KUKA KRL program: EPS_2_25694_LG05A_A_20260223033046.src

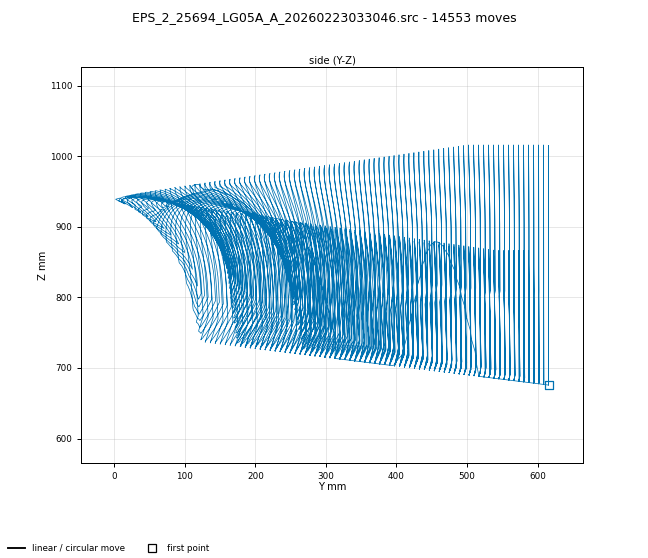
[picture p0: tool path of EPS_2_25694_LG05A_A_20260223033046.src, 14553 of 14555 moves have a stored position in this frame; points joined in program order, loops and branches not executed]
&ACCESS RVP
&REL 4
&COMMENT QRS 19112012
&PARAM EDITMASK = *
DEF PART()
EXT BAS (BAS_COMMAND :IN,REAL :IN )
INT I
BAS (#INITMOV,0 )

;KUKA QRS Post kuka4.cps  Date:22-06-2017 !

File_ID=3044

QRS_PRE_INIT()

;Init var - Until changes are made in qrs_pre_init
Outlet_Square_prg=0
Inlet_1_Square_prg=0
Inlet_2_Square_prg=0
Inlet_3_Square_prg=0
Inlet_4_Square_prg=0
Inlet_5_Square_prg=0

Outlet_1={X 0.000, Y 502.870, Z 915.500, B 0.000, E1 0.000 }
Inlet_1={X 0.000, Y 543.190, Z 350.500, B 0.000, E1 155.000 }
Inlet_2={X 0.000, Y 517.510, Z 710.500, B 0.000, E1 257.000 }
Outlet_1_type=201
Inlet_1_type=201
Inlet_2_type=201
;QRS#1=Sidecore dimensions
;QRS#2=200-8" PVC SDR 35
;QRS#3=200-8" PVC SDR 35
;QRS#4=200-8" PVC SDR 35
;QRS#5=
;QRS#6=
;QRS#7=
;QRS#8=
;QRS#9=12-08 PSX
;QRS#10=12-08 PSX
;QRS#11=12-08 PSX
;QRS#12=
;QRS#13=
;QRS#14=
;QRS#15=
;QRS#16=1220x127x1295 4,25'
;QRS#17=EPS Height
;QRS#18=1016
;QRS#19=*
;QRS#20= UPDATED VERSION 22-06-2017
;QRS#21=*
Outlet_Square=0100
Inlet_1_Square=0100
Inlet_2_Square=0100
Inlet_3_Square=0
Inlet_4_Square=0
Inlet_5_Square=0
Mill_Square=1
Outlet_Square_Prg=204
Inlet_1_Square_prg=204
Inlet_2_Square_prg=204

QRS_INIT()

$ADVANCE=5

; T1
PTP {E1 173.41,E2 173.41}
PTP {X 0,Y 615.487,A -85,B 0,C 180,E1 173.41,E2 173.41,E3 0,E4 0,E5 0,E6 0}
QRS_SPEED_INIT()
LIN {X 0,Y 615.487,Z 675.703,A -85,B 0,C 180,E1 173.41,E2 173.41,E3 0,E4 0,E5 0,E6 0} C_VEL
LIN {X 0,Y 615.494,Z 675.684,A -85,B 0,C 180,E1 170.801,E2 170.801} C_VEL
LIN {X 0,Y 615.457,Z 675.687,A -85,B 0,C 180,E1 168.138,E2 168.138} C_VEL
LIN {X 0,Y 615.465,Z 675.696,A -85,B 0,C 180,E1 165.45,E2 165.45} C_VEL
LIN {X 0,Y 615.489,Z 675.691,A -85,B 0,C 180,E1 162.729,E2 162.729} C_VEL
LIN {X 0,Y 615.462,Z 675.686,A -85,B 0,C 180,E1 159.966,E2 159.966} C_VEL
LIN {X 0,Y 615.452,Z 675.689,A -85,B 0,C 180,E1 157.659,E2 157.659} C_VEL
LIN {X 0,Y 615.47,Z 675.697,A -85,B 0,C 180,E1 155.007,E2 155.007} C_VEL
LIN {X 0,Y 615.484,Z 675.685,A -85,B 0,C 180,E1 152.084,E2 152.084} C_VEL
LIN {X 0,Y 615.481,Z 675.683,A -85,B 0,C 180,E1 149.839,E2 149.839} C_VEL
LIN {X 0,Y 615.46,Z 675.686,A -85,B 0,C 180,E1 147.541,E2 147.541} C_VEL
LIN {X 0,Y 615.448,Z 675.69,A -85,B 0,C 180,E1 145.182,E2 145.182} C_VEL
LIN {X 0,Y 615.456,Z 675.694,A -85,B 0,C 180,E1 142.755,E2 142.755} C_VEL
LIN {X 0,Y 615.49,Z 675.691,A -85,B 0,C 180,E1 139.909,E2 139.909} C_VEL
LIN {X 0,Y 615.497,Z 675.684,A -85,B 0,C 180,E1 137.647,E2 137.647} C_VEL
LIN {X 0,Y 615.449,Z 675.689,A -85,B 0,C 180,E1 134.927,E2 134.927} C_VEL
LIN {X 0,Y 615.476,Z 675.699,A -85,B 0,C 180,E1 132.078,E2 132.078} C_VEL
LIN {X 0,Y 615.466,Z 675.686,A -85,B 0,C 180,E1 129.059,E2 129.059} C_VEL
LIN {X 0,Y 615.496,Z 675.783,A -85,B 0,C 180,E1 127.719,E2 127.719} C_VEL
LIN {X 0,Y 615.495,Z 676.753,A -85,B 0,C 180,E1 127.575,E2 127.575} C_VEL
LIN {X 0,Y 615.499,Z 708.482,A -85,B 0,C 180,E1 127.183,E2 127.183} C_VEL
LIN {X 0,Y 615.497,Z 761.445,A -85,B 0,C 180,E1 126.551,E2 126.551} C_VEL
LIN {X 0,Y 615.5,Z 774.268,A -85,B 0,C 180,E1 126.275,E2 126.275} C_VEL
LIN {X 0,Y 615.5,Z 785.845,A -85,B 0,C 180,E1 125.908,E2 125.908} C_VEL
LIN {X 0,Y 615.495,Z 798.517,A -85,B 0,C 180,E1 125.363,E2 125.363} C_VEL
LIN {X 0,Y 615.485,Z 810.253,A -85,B 0,C 180,E1 124.7,E2 124.7} C_VEL
LIN {X 0,Y 615.497,Z 821.428,A -85,B 0,C 180,E1 123.898,E2 123.898} C_VEL
LIN {X 0,Y 615.497,Z 828.942,A -85,B 0,C 180,E1 123.234,E2 123.234} C_VEL
LIN {X 0,Y 615.496,Z 837.643,A -85,B 0,C 180,E1 122.331,E2 122.331} C_VEL
LIN {X 0,Y 615.493,Z 844.95,A -85,B 0,C 180,E1 121.385,E2 121.385} C_VEL
LIN {X 0,Y 615.495,Z 851.375,A -85,B 0,C 180,E1 120.348,E2 120.348} C_VEL
LIN {X 0,Y 615.498,Z 856.021,A -85,B 0,C 180,E1 119.404,E2 119.404} C_VEL
LIN {X 0,Y 615.496,Z 859.685,A -85,B 0,C 180,E1 118.451,E2 118.451} C_VEL
LIN {X 0,Y 615.496,Z 863.106,A -85,B 0,C 180,E1 117.175,E2 117.175} C_VEL
LIN {X 0,Y 615.493,Z 864.37,A -85,B 0,C 180,E1 116.443,E2 116.443} C_VEL
LIN {X 0,Y 615.496,Z 865.202,A -85,B 0,C 180,E1 115.569,E2 115.569} C_VEL
LIN {X 0,Y 615.494,Z 865.386,A -85,B 0,C 180,E1 114.99,E2 114.99} C_VEL
LIN {X 0,Y 615.496,Z 864.968,A -85,B 0,C 180,E1 114.009,E2 114.009} C_VEL
LIN {X 0,Y 615.496,Z 863.341,A -85,B 0,C 180,E1 112.843,E2 112.843} C_VEL
LIN {X 0,Y 615.495,Z 860.72,A -85,B 0,C 180,E1 111.782,E2 111.782} C_VEL
LIN {X 0,Y 615.497,Z 856.247,A -85,B 0,C 180,E1 110.558,E2 110.558} C_VEL
LIN {X 0,Y 615.496,Z 850.128,A -85,B 0,C 180,E1 109.336,E2 109.336} C_VEL
LIN {X 0,Y 615.494,Z 843.188,A -85,B 0,C 180,E1 108.28,E2 108.28} C_VEL
LIN {X 0,Y 615.498,Z 834.872,A -85,B 0,C 180,E1 107.269,E2 107.269} C_VEL
LIN {X 0,Y 615.498,Z 824.879,A -85,B 0,C 180,E1 106.3,E2 106.3} C_VEL
LIN {X 0,Y 615.491,Z 814.314,A -85,B 0,C 180,E1 105.479,E2 105.479} C_VEL
LIN {X 0,Y 615.488,Z 803.371,A -85,B 0,C 180,E1 104.802,E2 104.802} C_VEL
LIN {X 0,Y 615.498,Z 791.85,A -85,B 0,C 180,E1 104.241,E2 104.241} C_VEL
LIN {X 0,Y 615.496,Z 779.587,A -85,B 0,C 180,E1 103.789,E2 103.789} C_VEL
LIN {X 0,Y 615.498,Z 766.533,A -85,B 0,C 180,E1 103.452,E2 103.452} C_VEL
LIN {X 0,Y 615.5,Z 750.675,A -85,B 0,C 180,E1 103.221,E2 103.221} C_VEL
LIN {X 0,Y 615.498,Z 676.849,A -85,B 0,C 180,E1 102.34,E2 102.34} C_VEL
LIN {X 0,Y 615.493,Z 675.917,A -85,B 0,C 180,E1 102.236,E2 102.236} C_VEL
LIN {X 0,Y 615.473,Z 675.691,A -85,B 0,C 180,E1 100.526,E2 100.526} C_VEL
LIN {X 0,Y 615.478,Z 675.7,A -85,B 0,C 180,E1 97.875,E2 97.875} C_VEL
LIN {X 0,Y 615.428,Z 675.696,A -85,B 0,C 180,E1 95.241,E2 95.241} C_VEL
LIN {X 0,Y 615.432,Z 675.697,A -85,B 0,C 180,E1 93.272,E2 93.272} C_VEL
LIN {X 0,Y 615.439,Z 675.697,A -85,B 0,C 180,E1 91.308,E2 91.308} C_VEL
LIN {X 0,Y 615.447,Z 675.698,A -85,B 0,C 180,E1 89.345,E2 89.345} C_VEL
LIN {X 0,Y 615.457,Z 675.698,A -85,B 0,C 180,E1 87.381,E2 87.381} C_VEL
LIN {X 0,Y 615.422,Z 675.696,A -85,B 0,C 180,E1 84.757,E2 84.757} C_VEL
LIN {X 0,Y 615.424,Z 675.696,A -85,B 0,C 180,E1 82.783,E2 82.783} C_VEL
LIN {X 0,Y 615.426,Z 675.697,A -85,B 0,C 180,E1 80.799,E2 80.799} C_VEL
LIN {X 0,Y 615.429,Z 675.697,A -85,B 0,C 180,E1 78.805,E2 78.805} C_VEL
LIN {X 0,Y 615.429,Z 675.698,A -85,B 0,C 180,E1 76.797,E2 76.797} C_VEL
LIN {X 0,Y 615.435,Z 675.698,A -85,B 0,C 180,E1 74.772,E2 74.772} C_VEL
LIN {X 0,Y 615.436,Z 675.698,A -85,B 0,C 180,E1 72.727,E2 72.727} C_VEL
LIN {X 0,Y 615.435,Z 675.698,A -85,B 0,C 180,E1 70.659,E2 70.659} C_VEL
LIN {X 0,Y 615.433,Z 675.698,A -85,B 0,C 180,E1 68.565,E2 68.565} C_VEL
LIN {X 0,Y 615.427,Z 675.698,A -85,B 0,C 180,E1 66.44,E2 66.44} C_VEL
LIN {X 0,Y 615.421,Z 675.698,A -85,B 0,C 180,E1 64.28,E2 64.28} C_VEL
LIN {X 0,Y 615.417,Z 675.697,A -85,B 0,C 180,E1 62.081,E2 62.081} C_VEL
LIN {X 0,Y 615.415,Z 675.697,A -85,B 0,C 180,E1 59.835,E2 59.835} C_VEL
LIN {X 0,Y 615.425,Z 675.696,A -85,B 0,C 180,E1 57.538,E2 57.538} C_VEL
LIN {X 0,Y 615.449,Z 675.695,A -85,B 0,C 180,E1 55.182,E2 55.182} C_VEL
LIN {X 0,Y 615.489,Z 675.697,A -85,B 0,C 180,E1 52.757,E2 52.757} C_VEL
LIN {X 0,Y 615.425,Z 675.698,A -85,B 0,C 180,E1 49.918,E2 49.918} C_VEL
LIN {X 0,Y 615.415,Z 675.698,A -85,B 0,C 180,E1 47.64,E2 47.64} C_VEL
LIN {X 0,Y 615.439,Z 675.696,A -85,B 0,C 180,E1 44.926,E2 44.926} C_VEL
LIN {X 0,Y 615.467,Z 675.699,A -85,B 0,C 180,E1 42.077,E2 42.077} C_VEL
LIN {X 0,Y 615.436,Z 675.699,A -85,B 0,C 180,E1 39.755,E2 39.755} C_VEL
LIN {X 0,Y 615.41,Z 675.698,A -85,B 0,C 180,E1 37.248,E2 37.248} C_VEL
LIN {X 0,Y 615.428,Z 675.697,A -85,B 0,C 180,E1 34.691,E2 34.691} C_VEL
LIN {X 0,Y 615.46,Z 675.696,A -85,B 0,C 180,E1 32.325,E2 32.325} C_VEL
LIN {X 0,Y 615.432,Z 675.699,A -85,B 0,C 180,E1 29.409,E2 29.409} C_VEL
LIN {X 0,Y 615.412,Z 675.699,A -85,B 0,C 180,E1 27.03,E2 27.03} C_VEL
LIN {X 0,Y 615.499,Z 675.896,A -85,B 0,C 180,E1 25.679,E2 25.679} C_VEL
LIN {X 0,Y 615.5,Z 676.846,A -85,B 0,C 180,E1 25.57,E2 25.57} C_VEL
LIN {X 0,Y 615.495,Z 761.983,A -85,B 0,C 180,E1 24.541,E2 24.541} C_VEL
LIN {X 0,Y 615.498,Z 775.58,A -85,B 0,C 180,E1 24.239,E2 24.239} C_VEL
LIN {X 0,Y 615.497,Z 787.695,A -85,B 0,C 180,E1 23.839,E2 23.839} C_VEL
LIN {X 0,Y 615.493,Z 799.977,A -85,B 0,C 180,E1 23.289,E2 23.289} C_VEL
LIN {X 0,Y 615.485,Z 811.851,A -85,B 0,C 180,E1 22.595,E2 22.595} C_VEL
LIN {X 0,Y 615.498,Z 821.768,A -85,B 0,C 180,E1 21.872,E2 21.872} C_VEL
LIN {X 0,Y 615.499,Z 830.51,A -85,B 0,C 180,E1 21.081,E2 21.081} C_VEL
LIN {X 0,Y 615.496,Z 837.947,A -85,B 0,C 180,E1 20.295,E2 20.295} C_VEL
LIN {X 0,Y 615.497,Z 845.264,A -85,B 0,C 180,E1 19.338,E2 19.338} C_VEL
LIN {X 0,Y 615.498,Z 851.739,A -85,B 0,C 180,E1 18.281,E2 18.281} C_VEL
LIN {X 0,Y 615.495,Z 856.597,A -85,B 0,C 180,E1 17.27,E2 17.27} C_VEL
LIN {X 0,Y 615.495,Z 859.748,A -85,B 0,C 180,E1 16.431,E2 16.431} C_VEL
LIN {X 0,Y 615.496,Z 862.997,A -85,B 0,C 180,E1 15.226,E2 15.226} C_VEL
LIN {X 0,Y 615.494,Z 864.223,A -85,B 0,C 180,E1 14.549,E2 14.549} C_VEL
LIN {X 0,Y 615.494,Z 864.987,A -85,B 0,C 180,E1 13.874,E2 13.874} C_VEL
LIN {X 0,Y 615.495,Z 865.294,A -85,B 0,C 180,E1 12.53,E2 12.53} C_VEL
LIN {X 0,Y 615.495,Z 864.834,A -85,B 0,C 180,E1 11.861,E2 11.861} C_VEL
LIN {X 0,Y 615.494,Z 863.432,A -85,B 0,C 180,E1 10.888,E2 10.888} C_VEL
LIN {X 0,Y 615.498,Z 859.912,A -85,B 0,C 180,E1 9.53,E2 9.53} C_VEL
LIN {X 0,Y 615.495,Z 856.155,A -85,B 0,C 180,E1 8.537,E2 8.537} C_VEL
LIN {X 0,Y 615.497,Z 851.282,A -85,B 0,C 180,E1 7.546,E2 7.546} C_VEL
LIN {X 0,Y 615.488,Z 845.163,A -85,B 0,C 180,E1 6.557,E2 6.557} C_VEL
LIN {X 0,Y 615.498,Z 837.565,A -85,B 0,C 180,E1 5.57,E2 5.57} C_VEL
LIN {X 0,Y 615.497,Z 828.01,A -85,B 0,C 180,E1 4.585,E2 4.585} C_VEL
LIN {X 0,Y 615.5,Z 818.276,A -85,B 0,C 180,E1 3.765,E2 3.765} C_VEL
LIN {X 0,Y 615.492,Z 807.277,A -85,B 0,C 180,E1 3.027,E2 3.027} C_VEL
LIN {X 0,Y 615.498,Z 796.564,A -85,B 0,C 180,E1 2.454,E2 2.454} C_VEL
LIN {X 0,Y 615.5,Z 784.792,A -85,B 0,C 180,E1 1.963,E2 1.963} C_VEL
LIN {X 0,Y 615.498,Z 772.808,A -85,B 0,C 180,E1 1.595,E2 1.595} C_VEL
LIN {X 0,Y 615.499,Z 760.801,A -85,B 0,C 180,E1 1.35,E2 1.35} C_VEL
LIN {X 0,Y 615.497,Z 677.006,A -85,B 0,C 180,E1 0.348,E2 0.348} C_VEL
LIN {X 0,Y 615.498,Z 675.959,A -85,B 0,C 180,E1 0.245,E2 0.245} C_VEL
LIN {X 0,Y 615.469,Z 675.686,A -85,B 0,C 180,E1 -0.654,E2 -0.654} C_VEL
LIN {X 0,Y 615.489,Z 675.682,A -85,B 0,C 180,E1 -3.273,E2 -3.273} C_VEL
LIN {X 0,Y 615.488,Z 675.696,A -85,B 0,C 180,E1 -5.898,E2 -5.898} C_VEL
LIN {X 0,Y 615.471,Z 675.693,A -85,B 0,C 180,E1 -8.537,E2 -8.537} C_VEL
LIN {X 0,Y 615.483,Z 675.681,A -85,B 0,C 180,E1 -11.193,E2 -11.193} C_VEL
LIN {X 0,Y 615.482,Z 675.69,A -85,B 0,C 180,E1 -13.928,E2 -13.928} C_VEL
LIN {X 0,Y 615.48,Z 675.697,A -85,B 0,C 180,E1 -16.587,E2 -16.587} C_VEL
LIN {X 0,Y 615.474,Z 675.684,A -85,B 0,C 180,E1 -19.338,E2 -19.338} C_VEL
LIN {X 0,Y 615.482,Z 675.689,A -85,B 0,C 180,E1 -22.137,E2 -22.137} C_VEL
LIN {X 0,Y 615.473,Z 675.694,A -85,B 0,C 180,E1 -24.992,E2 -24.992} C_VEL
LIN {X 0,Y 615.468,Z 675.692,A -85,B 0,C 180,E1 -27.178,E2 -27.178} C_VEL
LIN {X 0,Y 615.481,Z 675.682,A -85,B 0,C 180,E1 -29.792,E2 -29.792} C_VEL
LIN {X 0,Y 615.481,Z 675.688,A -85,B 0,C 180,E1 -32.458,E2 -32.458} C_VEL
LIN {X 0,Y 615.488,Z 675.696,A -85,B 0,C 180,E1 -34.815,E2 -34.815} C_VEL
LIN {X 0,Y 615.479,Z 675.698,A -85,B 0,C 180,E1 -37.243,E2 -37.243} C_VEL
LIN {X 0,Y 615.475,Z 675.683,A -85,B 0,C 180,E1 -40.087,E2 -40.087} C_VEL
LIN {X 0,Y 615.487,Z 675.695,A -85,B 0,C 180,E1 -43.046,E2 -43.046} C_VEL
LIN {X 0,Y 615.466,Z 675.688,A -85,B 0,C 180,E1 -46.005,E2 -46.005} C_VEL
LIN {X 0,Y 615.485,Z 675.686,A -85,B 0,C 180,E1 -48.906,E2 -48.906} C_VEL
LIN {X 0,Y 615.482,Z 675.689,A -85,B 0,C 180,E1 -51.094,E2 -51.094} C_VEL
LIN {X 0,Y 615.484,Z 675.703,A -85,B 0,C 180,E1 -53.574,E2 -53.574} C_VEL
LIN {X 0,Y 615.473,Z 675.695,A -85,B 0,C 180,E1 -55.976,E2 -55.976} C_VEL
LIN {X 0,Y 615.464,Z 675.69,A -85,B 0,C 180,E1 -58.312,E2 -58.312} C_VEL
LIN {X 0,Y 615.467,Z 675.686,A -85,B 0,C 180,E1 -60.592,E2 -60.592} C_VEL
LIN {X 0,Y 615.485,Z 675.681,A -85,B 0,C 180,E1 -62.956,E2 -62.956} C_VEL
LIN {X 0,Y 615.497,Z 675.933,A -85,B 0,C 180,E1 -64.057,E2 -64.057} C_VEL
LIN {X 0,Y 615.472,Z 692.484,A -85,B 0,C 180,E1 -65.863,E2 -65.863} C_VEL
LIN {X 0,Y 615.448,Z 716.422,A -85,B 0,C 180,E1 -68.39,E2 -68.39} C_VEL
LIN {X 0,Y 615.482,Z 743.317,A -85,B 0,C 180,E1 -71.18,E2 -71.18} C_VEL
LIN {X 0,Y 615.458,Z 771.867,A -85,B 0,C 180,E1 -74.093,E2 -74.093} C_VEL
LIN {X 0,Y 615.477,Z 798.699,A -85,B 0,C 180,E1 -76.798,E2 -76.798} C_VEL
LIN {X 0,Y 615.495,Z 801.848,A -85,B 0,C 180,E1 -77.092,E2 -77.092} C_VEL
LIN {X 0,Y 615.483,Z 911.78,A -85,B 0,C 180,E1 -78.41,E2 -78.41} C_VEL
LIN {X 0,Y 615.498,Z 924.309,A -85,B 0,C 180,E1 -78.681,E2 -78.681} C_VEL
LIN {X 0,Y 615.496,Z 937.503,A -85,B 0,C 180,E1 -79.109,E2 -79.109} C_VEL
LIN {X 0,Y 615.493,Z 949.458,A -85,B 0,C 180,E1 -79.639,E2 -79.639} C_VEL
LIN {X 0,Y 615.483,Z 960.982,A -85,B 0,C 180,E1 -80.303,E2 -80.303} C_VEL
LIN {X 0,Y 615.499,Z 971.329,A -85,B 0,C 180,E1 -81.049,E2 -81.049} C_VEL
LIN {X 0,Y 615.497,Z 979.682,A -85,B 0,C 180,E1 -81.793,E2 -81.793} C_VEL
LIN {X 0,Y 615.498,Z 987.598,A -85,B 0,C 180,E1 -82.619,E2 -82.619} C_VEL
LIN {X 0,Y 615.491,Z 995.198,A -85,B 0,C 180,E1 -83.607,E2 -83.607} C_VEL
LIN {X 0,Y 615.498,Z 1002.199,A -85,B 0,C 180,E1 -84.758,E2 -84.758} C_VEL
LIN {X 0,Y 615.493,Z 1006.847,A -85,B 0,C 180,E1 -85.743,E2 -85.743} C_VEL
LIN {X 0,Y 615.494,Z 1010.396,A -85,B 0,C 180,E1 -86.726,E2 -86.726} C_VEL
LIN {X 0,Y 615.497,Z 1012.23,A -85,B 0,C 180,E1 -87.381,E2 -87.381} C_VEL
LIN {X 0,Y 615.497,Z 1013.607,A -85,B 0,C 180,E1 -88.036,E2 -88.036} C_VEL
LIN {X 0,Y 615.496,Z 1015.173,A -85,B 0,C 180,E1 -89.345,E2 -89.345} C_VEL
LIN {X 0,Y 615.494,Z 1015.389,A -85,B 0,C 180,E1 -89.999,E2 -89.999} C_VEL
LIN {X 0,Y 615.495,Z 1014.581,A -85,B 0,C 180,E1 -91.308,E2 -91.308} C_VEL
LIN {X 0,Y 615.497,Z 1013.61,A -85,B 0,C 180,E1 -91.962,E2 -91.962} C_VEL
LIN {X 0,Y 615.497,Z 1012.235,A -85,B 0,C 180,E1 -92.617,E2 -92.617} C_VEL
LIN {X 0,Y 615.496,Z 1009.353,A -85,B 0,C 180,E1 -93.6,E2 -93.6} C_VEL
LIN {X 0,Y 615.498,Z 1005.446,A -85,B 0,C 180,E1 -94.583,E2 -94.583} C_VEL
LIN {X 0,Y 615.499,Z 1000.41,A -85,B 0,C 180,E1 -95.569,E2 -95.569} C_VEL
LIN {X 0,Y 615.49,Z 993.913,A -85,B 0,C 180,E1 -96.578,E2 -96.578} C_VEL
LIN {X 0,Y 615.497,Z 986.142,A -85,B 0,C 180,E1 -97.544,E2 -97.544} C_VEL
LIN {X 0,Y 615.498,Z 976.269,A -85,B 0,C 180,E1 -98.535,E2 -98.535} C_VEL
LIN {X 0,Y 615.495,Z 965.88,A -85,B 0,C 180,E1 -99.363,E2 -99.363} C_VEL
LIN {X 0,Y 615.482,Z 955.594,A -85,B 0,C 180,E1 -100.027,E2 -100.027} C_VEL
LIN {X 0,Y 615.497,Z 944.112,A -85,B 0,C 180,E1 -100.617,E2 -100.617} C_VEL
LIN {X 0,Y 615.499,Z 932.285,A -85,B 0,C 180,E1 -101.079,E2 -101.079} C_VEL
LIN {X 0,Y 615.494,Z 919.286,A -85,B 0,C 180,E1 -101.442,E2 -101.442} C_VEL
LIN {X 0,Y 615.479,Z 906.029,A -85,B 0,C 180,E1 -101.672,E2 -101.672} C_VEL
LIN {X 0,Y 615.495,Z 801.887,A -85,B 0,C 180,E1 -102.906,E2 -102.906} C_VEL
LIN {X 0,Y 615.439,Z 776.921,A -85,B 0,C 180,E1 -105.396,E2 -105.396} C_VEL
LIN {X 0,Y 615.495,Z 751.738,A -85,B 0,C 180,E1 -107.956,E2 -107.956} C_VEL
LIN {X 0,Y 615.492,Z 724.847,A -85,B 0,C 180,E1 -110.729,E2 -110.729} C_VEL
LIN {X 0,Y 615.444,Z 699.632,A -85,B 0,C 180,E1 -113.379,E2 -113.379} C_VEL
LIN {X 0,Y 615.494,Z 676.165,A -85,B 0,C 180,E1 -115.896,E2 -115.896} C_VEL
LIN {X 0,Y 615.498,Z 675.721,A -85,B 0,C 180,E1 -116.078,E2 -116.078} C_VEL
LIN {X 0,Y 615.485,Z 675.687,A -85,B 0,C 180,E1 -118.657,E2 -118.657} C_VEL
LIN {X 0,Y 615.482,Z 675.682,A -85,B 0,C 180,E1 -121.085,E2 -121.085} C_VEL
LIN {X 0,Y 615.467,Z 675.686,A -85,B 0,C 180,E1 -123.531,E2 -123.531} C_VEL
LIN {X 0,Y 615.462,Z 675.69,A -85,B 0,C 180,E1 -125.83,E2 -125.83} C_VEL
LIN {X 0,Y 615.462,Z 675.693,A -85,B 0,C 180,E1 -128.069,E2 -128.069} C_VEL
LIN {X 0,Y 615.488,Z 675.703,A -85,B 0,C 180,E1 -130.605,E2 -130.605} C_VEL
LIN {X 0,Y 615.489,Z 675.684,A -85,B 0,C 180,E1 -133.243,E2 -133.243} C_VEL
LIN {X 0,Y 615.463,Z 675.687,A -85,B 0,C 180,E1 -136.003,E2 -136.003} C_VEL
LIN {X 0,Y 615.468,Z 675.694,A -85,B 0,C 180,E1 -138.524,E2 -138.524} C_VEL
LIN {X 0,Y 615.492,Z 675.697,A -85,B 0,C 180,E1 -141.096,E2 -141.096} C_VEL
LIN {X 0,Y 615.489,Z 675.685,A -85,B 0,C 180,E1 -143.575,E2 -143.575} C_VEL
LIN {X 0,Y 615.487,Z 675.681,A -85,B 0,C 180,E1 -145.978,E2 -145.978} C_VEL
LIN {X 0,Y 615.466,Z 675.685,A -85,B 0,C 180,E1 -148.313,E2 -148.313} C_VEL
LIN {X 0,Y 615.459,Z 675.688,A -85,B 0,C 180,E1 -150.592,E2 -150.592} C_VEL
LIN {X 0,Y 615.463,Z 675.693,A -85,B 0,C 180,E1 -152.957,E2 -152.957} C_VEL
LIN {X 0,Y 615.489,Z 675.693,A -85,B 0,C 180,E1 -155.728,E2 -155.728} C_VEL
LIN {X 0,Y 615.471,Z 675.684,A -85,B 0,C 180,E1 -158.568,E2 -158.568} C_VEL
LIN {X 0,Y 615.469,Z 675.684,A -85,B 0,C 180,E1 -160.661,E2 -160.661} C_VEL
LIN {X 0,Y 615.465,Z 675.695,A -85,B 0,C 180,E1 -163.413,E2 -163.413} C_VEL
LIN {X 0,Y 615.488,Z 675.692,A -85,B 0,C 180,E1 -166.126,E2 -166.126} C_VEL
LIN {X 0,Y 615.479,Z 675.682,A -85,B 0,C 180,E1 -168.807,E2 -168.807} C_VEL
LIN {X 0,Y 615.456,Z 675.691,A -85,B 0,C 180,E1 -171.463,E2 -171.463} C_VEL
LIN {X 0,Y 615.494,Z 675.699,A -85,B 0,C 180,E1 -174.102,E2 -174.102} C_VEL
LIN {X 0,Y 615.492,Z 675.685,A -85,B 0,C 180,E1 -176.727,E2 -176.727} C_VEL
LIN {X 0,Y 615.461,Z 675.686,A -85,B 0,C 180,E1 -179.346,E2 -179.346} C_VEL
LIN {X 0,Y 615.458,Z 675.693,A -85,B 0,C 180,E1 -181.963,E2 -181.963} C_VEL
LIN {X 0,Y 615.497,Z 675.698,A -85,B 0,C 180,E1 -184.585,E2 -184.585} C_VEL
LIN {X 0,Y 615.487,Z 675.703,A -85,B 0,C 180,E1 -186.59,E2 -186.59} C_VEL
LIN {X 0,Y 614.814,Z 675.833,A -85,B 0,C 180,E1 -187.136,E2 -187.136} C_VEL
LIN {X 0,Y 611.988,Z 676.247,A -85,B 0,C 180,E1 -188.022,E2 -188.022} C_VEL
LIN {X 0,Y 609.594,Z 676.558,A -85,B 0,C 180,E1 -188.734,E2 -188.734} C_VEL
LIN {X 0,Y 608.548,Z 676.677,A -85,B 0,C 180,E1 -189.284,E2 -189.284} C_VEL
LIN {X 0,Y 608.452,Z 676.687,A -85,B 0,C 180,E1 -189.47,E2 -189.47} C_VEL
LIN {X 0,Y 608.437,Z 676.689,A -85,B 0,C 180,E1 -192,E2 -192} C_VEL
LIN {X 0,Y 608.461,Z 676.694,A -85,B 0,C 180,E1 -194.721,E2 -194.721} C_VEL
LIN {X 0,Y 608.447,Z 676.69,A -85,B 0,C 180,E1 -197.477,E2 -197.477} C_VEL
LIN {X 0,Y 608.435,Z 676.689,A -85,B 0,C 180,E1 -200.275,E2 -200.275} C_VEL
LIN {X 0,Y 608.447,Z 676.688,A -85,B 0,C 180,E1 -202.477,E2 -202.477} C_VEL
LIN {X 0,Y 608.446,Z 676.698,A -85,B 0,C 180,E1 -205.301,E2 -205.301} C_VEL
LIN {X 0,Y 608.442,Z 676.696,A -85,B 0,C 180,E1 -207.519,E2 -207.519} C_VEL
LIN {X 0,Y 608.451,Z 676.686,A -85,B 0,C 180,E1 -210.546,E2 -210.546} C_VEL
LIN {X 0,Y 608.437,Z 676.689,A -85,B 0,C 180,E1 -212.881,E2 -212.881} C_VEL
LIN {X 0,Y 608.434,Z 676.694,A -85,B 0,C 180,E1 -215.279,E2 -215.279} C_VEL
LIN {X 0,Y 608.466,Z 676.687,A -85,B 0,C 180,E1 -218.242,E2 -218.242} C_VEL
LIN {X 0,Y 608.419,Z 676.692,A -85,B 0,C 180,E1 -221.18,E2 -221.18} C_VEL
LIN {X 0,Y 608.466,Z 676.696,A -85,B 0,C 180,E1 -223.87,E2 -223.87} C_VEL
LIN {X 0,Y 608.464,Z 676.686,A -85,B 0,C 180,E1 -226.692,E2 -226.692} C_VEL
LIN {X 0,Y 608.443,Z 676.688,A -85,B 0,C 180,E1 -228.824,E2 -228.824} C_VEL
LIN {X 0,Y 608.448,Z 676.691,A -85,B 0,C 180,E1 -231.763,E2 -231.763} C_VEL
LIN {X 0,Y 608.505,Z 676.96,A -85,B 0,C 180,E1 -232.221,E2 -232.221} C_VEL
LIN {X 0,Y 608.596,Z 677.93,A -85,B 0,C 180,E1 -232.305,E2 -232.305} C_VEL
LIN {X 0,Y 608.563,Z 762.201,A -85,B 0,C 180,E1 -233.327,E2 -233.327} C_VEL
LIN {X 0,Y 608.547,Z 775.37,A -85,B 0,C 180,E1 -233.621,E2 -233.621} C_VEL
LIN {X 0,Y 608.526,Z 787.298,A -85,B 0,C 180,E1 -234.015,E2 -234.015} C_VEL
LIN {X 0,Y 608.518,Z 798.871,A -85,B 0,C 180,E1 -234.526,E2 -234.526} C_VEL
LIN {X 0,Y 608.474,Z 810.468,A -85,B 0,C 180,E1 -235.188,E2 -235.188} C_VEL
LIN {X 0,Y 608.472,Z 820.84,A -85,B 0,C 180,E1 -235.931,E2 -235.931} C_VEL
LIN {X 0,Y 608.475,Z 828.838,A -85,B 0,C 180,E1 -236.629,E2 -236.629} C_VEL
LIN {X 0,Y 608.473,Z 837.054,A -85,B 0,C 180,E1 -237.477,E2 -237.477} C_VEL
LIN {X 0,Y 608.453,Z 845.023,A -85,B 0,C 180,E1 -238.49,E2 -238.49} C_VEL
LIN {X 0,Y 608.444,Z 851.11,A -85,B 0,C 180,E1 -239.455,E2 -239.455} C_VEL
LIN {X 0,Y 608.433,Z 856.778,A -85,B 0,C 180,E1 -240.601,E2 -240.601} C_VEL
LIN {X 0,Y 608.439,Z 860.956,A -85,B 0,C 180,E1 -241.734,E2 -241.734} C_VEL
LIN {X 0,Y 608.438,Z 863.698,A -85,B 0,C 180,E1 -242.801,E2 -242.801} C_VEL
LIN {X 0,Y 608.421,Z 865.47,A -85,B 0,C 180,E1 -243.965,E2 -243.965} C_VEL
LIN {X 0,Y 608.438,Z 865.925,A -85,B 0,C 180,E1 -244.7,E2 -244.7} C_VEL
LIN {X 0,Y 608.422,Z 865.676,A -85,B 0,C 180,E1 -245.86,E2 -245.86} C_VEL
LIN {X 0,Y 608.433,Z 864.458,A -85,B 0,C 180,E1 -246.877,E2 -246.877} C_VEL
LIN {X 0,Y 608.433,Z 863.038,A -85,B 0,C 180,E1 -247.594,E2 -247.594} C_VEL
LIN {X 0,Y 608.439,Z 859.972,A -85,B 0,C 180,E1 -248.664,E2 -248.664} C_VEL
LIN {X 0,Y 608.443,Z 855.758,A -85,B 0,C 180,E1 -249.726,E2 -249.726} C_VEL
LIN {X 0,Y 608.445,Z 849.205,A -85,B 0,C 180,E1 -250.956,E2 -250.956} C_VEL
LIN {X 0,Y 608.462,Z 842.051,A -85,B 0,C 180,E1 -252.004,E2 -252.004} C_VEL
LIN {X 0,Y 608.458,Z 834.756,A -85,B 0,C 180,E1 -252.871,E2 -252.871} C_VEL
LIN {X 0,Y 608.47,Z 825.459,A -85,B 0,C 180,E1 -253.774,E2 -253.774} C_VEL
LIN {X 0,Y 608.482,Z 815.022,A -85,B 0,C 180,E1 -254.596,E2 -254.596} C_VEL
LIN {X 0,Y 608.506,Z 804.188,A -85,B 0,C 180,E1 -255.281,E2 -255.281} C_VEL
LIN {X 0,Y 608.525,Z 792.068,A -85,B 0,C 180,E1 -255.88,E2 -255.88} C_VEL
LIN {X 0,Y 608.526,Z 779.478,A -85,B 0,C 180,E1 -256.348,E2 -256.348} C_VEL
LIN {X 0,Y 608.546,Z 766.239,A -85,B 0,C 180,E1 -256.689,E2 -256.689} C_VEL
LIN {X 0,Y 608.564,Z 750.129,A -85,B 0,C 180,E1 -256.923,E2 -256.923} C_VEL
LIN {X 0,Y 608.613,Z 677.735,A -85,B 0,C 180,E1 -257.793,E2 -257.793} C_VEL
LIN {X 0,Y 608.489,Z 676.763,A -85,B 0,C 180,E1 -257.917,E2 -257.917} C_VEL
LIN {X 0,Y 608.421,Z 676.691,A -85,B 0,C 180,E1 -260.695,E2 -260.695} C_VEL
LIN {X 0,Y 608.409,Z 676.693,A -85,B 0,C 180,E1 -262.701,E2 -262.701} C_VEL
LIN {X 0,Y 608.417,Z 676.693,A -85,B 0,C 180,E1 -264.699,E2 -264.699} C_VEL
LIN {X 0,Y 608.431,Z 676.689,A -85,B 0,C 180,E1 -267.353,E2 -267.353} C_VEL
LIN {X 0,Y 608.477,Z 676.69,A -85,B 0,C 180,E1 -270.001,E2 -270.001} C_VEL
LIN {X 0,Y 608.449,Z 676.692,A -85,B 0,C 180,E1 -272.649,E2 -272.649} C_VEL
LIN {X 0,Y 608.408,Z 676.692,A -85,B 0,C 180,E1 -275.303,E2 -275.303} C_VEL
LIN {X 0,Y 608.417,Z 676.693,A -85,B 0,C 180,E1 -277.969,E2 -277.969} C_VEL
LIN {X 0,Y 608.421,Z 676.695,A -85,B 0,C 180,E1 -280.93,E2 -280.93} C_VEL
LIN {X 0,Y 608.41,Z 676.693,A -85,B 0,C 180,E1 -283.359,E2 -283.359} C_VEL
LIN {X 0,Y 608.423,Z 676.691,A -85,B 0,C 180,E1 -285.408,E2 -285.408} C_VEL
LIN {X 0,Y 608.405,Z 676.693,A -85,B 0,C 180,E1 -287.479,E2 -287.479} C_VEL
LIN {X 0,Y 608.404,Z 676.693,A -85,B 0,C 180,E1 -289.573,E2 -289.573} C_VEL
LIN {X 0,Y 608.419,Z 676.691,A -85,B 0,C 180,E1 -291.694,E2 -291.694} C_VEL
LIN {X 0,Y 608.43,Z 676.693,A -85,B 0,C 180,E1 -294.573,E2 -294.573} C_VEL
LIN {X 0,Y 608.422,Z 676.694,A -85,B 0,C 180,E1 -297.52,E2 -297.52} C_VEL
LIN {X 0,Y 608.391,Z 676.694,A -85,B 0,C 180,E1 -299.958,E2 -299.958} C_VEL
LIN {X 0,Y 608.412,Z 676.692,A -85,B 0,C 180,E1 -302.514,E2 -302.514} C_VEL
LIN {X 0,Y 608.416,Z 676.701,A -85,B 0,C 180,E1 -305.28,E2 -305.28} C_VEL
LIN {X 0,Y 608.433,Z 676.694,A -85,B 0,C 180,E1 -307.75,E2 -307.75} C_VEL
LIN {X 0,Y 608.409,Z 676.692,A -85,B 0,C 180,E1 -310.324,E2 -310.324} C_VEL
LIN {X 0,Y 608.389,Z 676.695,A -85,B 0,C 180,E1 -312.326,E2 -312.326} C_VEL
LIN {X 0,Y 608.402,Z 676.693,A -85,B 0,C 180,E1 -314.802,E2 -314.802} C_VEL
LIN {X 0,Y 608.467,Z 676.696,A -85,B 0,C 180,E1 -317.666,E2 -317.666} C_VEL
LIN {X 0,Y 608.46,Z 676.696,A -85,B 0,C 180,E1 -319.697,E2 -319.697} C_VEL
LIN {X 0,Y 608.419,Z 676.695,A -85,B 0,C 180,E1 -322.25,E2 -322.25} C_VEL
LIN {X 0,Y 608.394,Z 676.694,A -85,B 0,C 180,E1 -324.719,E2 -324.719} C_VEL
LIN {X 0,Y 608.426,Z 676.692,A -85,B 0,C 180,E1 -327.484,E2 -327.484} C_VEL
LIN {X 0,Y 608.466,Z 676.694,A -85,B 0,C 180,E1 -330.22,E2 -330.22} C_VEL
LIN {X 0,Y 608.381,Z 676.695,A -85,B 0,C 180,E1 -333.222,E2 -333.222} C_VEL
LIN {X 0,Y 608.508,Z 676.892,A -85,B 0,C 180,E1 -334.209,E2 -334.209} C_VEL
LIN {X 0,Y 608.592,Z 678.051,A -85,B 0,C 180,E1 -334.309,E2 -334.309} C_VEL
LIN {X 0,Y 608.543,Z 761.782,A -85,B 0,C 180,E1 -335.319,E2 -335.319} C_VEL
LIN {X 0,Y 608.533,Z 774.704,A -85,B 0,C 180,E1 -335.603,E2 -335.603} C_VEL
LIN {X 0,Y 608.518,Z 786.494,A -85,B 0,C 180,E1 -335.985,E2 -335.985} C_VEL
LIN {X 0,Y 608.514,Z 798.699,A -85,B 0,C 180,E1 -336.518,E2 -336.518} C_VEL
LIN {X 0,Y 608.484,Z 810.248,A -85,B 0,C 180,E1 -337.174,E2 -337.174} C_VEL
LIN {X 0,Y 608.498,Z 821.111,A -85,B 0,C 180,E1 -337.953,E2 -337.953} C_VEL
LIN {X 0,Y 608.463,Z 829.186,A -85,B 0,C 180,E1 -338.664,E2 -338.664} C_VEL
LIN {X 0,Y 608.458,Z 838.077,A -85,B 0,C 180,E1 -339.593,E2 -339.593} C_VEL
LIN {X 0,Y 608.45,Z 845.791,A -85,B 0,C 180,E1 -340.605,E2 -340.605} C_VEL
LIN {X 0,Y 608.445,Z 851.691,A -85,B 0,C 180,E1 -341.562,E2 -341.562} C_VEL
LIN {X 0,Y 608.429,Z 856.443,A -85,B 0,C 180,E1 -342.523,E2 -342.523} C_VEL
LIN {X 0,Y 608.426,Z 860.166,A -85,B 0,C 180,E1 -343.486,E2 -343.486} C_VEL
LIN {X 0,Y 608.42,Z 863.247,A -85,B 0,C 180,E1 -344.593,E2 -344.593} C_VEL
LIN {X 0,Y 608.417,Z 864.565,A -85,B 0,C 180,E1 -345.278,E2 -345.278} C_VEL
LIN {X 0,Y 608.446,Z 865.501,A -85,B 0,C 180,E1 -345.994,E2 -345.994} C_VEL
LIN {X 0,Y 608.438,Z 865.912,A -85,B 0,C 180,E1 -346.643,E2 -346.643} C_VEL
LIN {X 0,Y 608.44,Z 865.578,A -85,B 0,C 180,E1 -348,E2 -348} C_VEL
LIN {X 0,Y 608.434,Z 864.145,A -85,B 0,C 180,E1 -349.065,E2 -349.065} C_VEL
LIN {X 0,Y 608.43,Z 860.949,A -85,B 0,C 180,E1 -350.358,E2 -350.358} C_VEL
LIN {X 0,Y 608.427,Z 857.317,A -85,B 0,C 180,E1 -351.363,E2 -351.363} C_VEL
LIN {X 0,Y 608.451,Z 852.572,A -85,B 0,C 180,E1 -352.367,E2 -352.367} C_VEL
LIN {X 0,Y 608.443,Z 845.681,A -85,B 0,C 180,E1 -353.502,E2 -353.502} C_VEL
LIN {X 0,Y 608.462,Z 837.781,A -85,B 0,C 180,E1 -354.532,E2 -354.532} C_VEL
LIN {X 0,Y 608.474,Z 828.148,A -85,B 0,C 180,E1 -355.528,E2 -355.528} C_VEL
LIN {X 0,Y 608.48,Z 818.307,A -85,B 0,C 180,E1 -356.358,E2 -356.358} C_VEL
LIN {X 0,Y 608.5,Z 807.196,A -85,B 0,C 180,E1 -357.103,E2 -357.103} C_VEL
LIN {X 0,Y 608.514,Z 796.387,A -85,B 0,C 180,E1 -357.683,E2 -357.683} C_VEL
LIN {X 0,Y 608.54,Z 784.486,A -85,B 0,C 180,E1 -358.18,E2 -358.18} C_VEL
LIN {X 0,Y 608.555,Z 772.298,A -85,B 0,C 180,E1 -358.552,E2 -358.552} C_VEL
LIN {X 0,Y 608.548,Z 758.368,A -85,B 0,C 180,E1 -358.821,E2 -358.821} C_VEL
LIN {X 0,Y 608.589,Z 677.729,A -85,B 0,C 180,E1 -359.793,E2 -359.793} C_VEL
LIN {X 0,Y 608.47,Z 676.768,A -85,B 0,C 180,E1 -359.917,E2 -359.917} C_VEL
LIN {X 0,Y 608.463,Z 676.686,A -85,B 0,C 180,E1 -362.648,E2 -362.648} C_VEL
LIN {X 0,Y 608.469,Z 676.685,A -85,B 0,C 180,E1 -365.302,E2 -365.302} C_VEL
LIN {X 0,Y 608.476,Z 676.692,A -85,B 0,C 180,E1 -367.967,E2 -367.967} C_VEL
LIN {X 0,Y 608.452,Z 676.69,A -85,B 0,C 180,E1 -370.65,E2 -370.65} C_VEL
LIN {X 0,Y 608.458,Z 676.686,A -85,B 0,C 180,E1 -373.357,E2 -373.357} C_VEL
LIN {X 0,Y 608.46,Z 676.691,A -85,B 0,C 180,E1 -376.094,E2 -376.094} C_VEL
LIN {X 0,Y 608.455,Z 676.69,A -85,B 0,C 180,E1 -378.87,E2 -378.87} C_VEL
LIN {X 0,Y 608.46,Z 676.686,A -85,B 0,C 180,E1 -381.692,E2 -381.692} C_VEL
LIN {X 0,Y 608.447,Z 676.697,A -85,B 0,C 180,E1 -384.571,E2 -384.571} C_VEL
LIN {X 0,Y 608.446,Z 676.691,A -85,B 0,C 180,E1 -387.2,E2 -387.2} C_VEL
LIN {X 0,Y 608.466,Z 676.685,A -85,B 0,C 180,E1 -389.97,E2 -389.97} C_VEL
LIN {X 0,Y 608.451,Z 676.698,A -85,B 0,C 180,E1 -392.88,E2 -392.88} C_VEL
LIN {X 0,Y 608.434,Z 676.695,A -85,B 0,C 180,E1 -395.278,E2 -395.278} C_VEL
LIN {X 0,Y 608.462,Z 676.686,A -85,B 0,C 180,E1 -397.747,E2 -397.747} C_VEL
LIN {X 0,Y 608.446,Z 676.687,A -85,B 0,C 180,E1 -400.327,E2 -400.327} C_VEL
LIN {X 0,Y 608.483,Z 676.694,A -85,B 0,C 180,E1 -403.309,E2 -403.309} C_VEL
LIN {X 0,Y 608.456,Z 676.686,A -85,B 0,C 180,E1 -406.128,E2 -406.128} C_VEL
LIN {X 0,Y 608.456,Z 676.688,A -85,B 0,C 180,E1 -408.823,E2 -408.823} C_VEL
LIN {X 0,Y 608.456,Z 676.693,A -85,B 0,C 180,E1 -411.761,E2 -411.761} C_VEL
LIN {X 0,Y 608.445,Z 676.692,A -85,B 0,C 180,E1 -413.955,E2 -413.955} C_VEL
LIN {X 0,Y 608.449,Z 676.688,A -85,B 0,C 180,E1 -416.327,E2 -416.327} C_VEL
LIN {X 0,Y 608.448,Z 676.687,A -85,B 0,C 180,E1 -418.733,E2 -418.733} C_VEL
LIN {X 0,Y 608.474,Z 676.688,A -85,B 0,C 180,E1 -421.38,E2 -421.38} C_VEL
LIN {X 0,Y 608.489,Z 676.877,A -85,B 0,C 180,E1 -423.85,E2 -423.85} C_VEL
LIN {X 0,Y 608.73,Z 680.067,A -85,B 0,C 180,E1 -424.229,E2 -424.229} C_VEL
LIN {X 0,Y 608.625,Z 702.974,A -85,B 0,C 180,E1 -426.702,E2 -426.702} C_VEL
LIN {X 0,Y 608.606,Z 730.295,A -85,B 0,C 180,E1 -429.598,E2 -429.598} C_VEL
LIN {X 0,Y 608.555,Z 756.766,A -85,B 0,C 180,E1 -432.352,E2 -432.352} C_VEL
LIN {X 0,Y 608.499,Z 783.662,A -85,B 0,C 180,E1 -435.108,E2 -435.108} C_VEL
LIN {X 0,Y 608.513,Z 801.915,A -85,B 0,C 180,E1 -436.941,E2 -436.941} C_VEL
LIN {X 0,Y 608.583,Z 839.839,A -85,B 0,C 180,E1 -437.409,E2 -437.409} C_VEL
LIN {X 0,Y 608.533,Z 911.896,A -85,B 0,C 180,E1 -438.275,E2 -438.275} C_VEL
LIN {X 0,Y 608.545,Z 925.183,A -85,B 0,C 180,E1 -438.571,E2 -438.571} C_VEL
LIN {X 0,Y 608.545,Z 938.322,A -85,B 0,C 180,E1 -439.009,E2 -439.009} C_VEL
LIN {X 0,Y 608.515,Z 949.617,A -85,B 0,C 180,E1 -439.518,E2 -439.518} C_VEL
LIN {X 0,Y 608.471,Z 961.183,A -85,B 0,C 180,E1 -440.19,E2 -440.19} C_VEL
LIN {X 0,Y 608.485,Z 971.582,A -85,B 0,C 180,E1 -440.945,E2 -440.945} C_VEL
LIN {X 0,Y 608.459,Z 979.99,A -85,B 0,C 180,E1 -441.698,E2 -441.698} C_VEL
LIN {X 0,Y 608.471,Z 987.952,A -85,B 0,C 180,E1 -442.533,E2 -442.533} C_VEL
LIN {X 0,Y 608.437,Z 995.295,A -85,B 0,C 180,E1 -443.486,E2 -443.486} C_VEL
LIN {X 0,Y 608.45,Z 1000.861,A -85,B 0,C 180,E1 -444.365,E2 -444.365} C_VEL
LIN {X 0,Y 608.432,Z 1005.946,A -85,B 0,C 180,E1 -445.361,E2 -445.361} C_VEL
LIN {X 0,Y 608.449,Z 1009.893,A -85,B 0,C 180,E1 -446.357,E2 -446.357} C_VEL
LIN {X 0,Y 608.425,Z 1012.807,A -85,B 0,C 180,E1 -447.351,E2 -447.351} C_VEL
LIN {X 0,Y 608.442,Z 1014.2,A -85,B 0,C 180,E1 -448.013,E2 -448.013} C_VEL
LIN {X 0,Y 608.438,Z 1015.783,A -85,B 0,C 180,E1 -449.337,E2 -449.337} C_VEL
LIN {X 0,Y 608.434,Z 1016,A -85,B 0,C 180,E1 -449.999,E2 -449.999} C_VEL
LIN {X 0,Y 608.448,Z 1015.185,A -85,B 0,C 180,E1 -451.323,E2 -451.323} C_VEL
LIN {X 0,Y 608.442,Z 1014.203,A -85,B 0,C 180,E1 -451.985,E2 -451.985} C_VEL
LIN {X 0,Y 608.425,Z 1012.812,A -85,B 0,C 180,E1 -452.647,E2 -452.647} C_VEL
LIN {X 0,Y 608.449,Z 1009.9,A -85,B 0,C 180,E1 -453.641,E2 -453.641} C_VEL
LIN {X 0,Y 608.432,Z 1005.954,A -85,B 0,C 180,E1 -454.637,E2 -454.637} C_VEL
LIN {X 0,Y 608.437,Z 999.883,A -85,B 0,C 180,E1 -455.8,E2 -455.8} C_VEL
LIN {X 0,Y 608.46,Z 993.243,A -85,B 0,C 180,E1 -456.798,E2 -456.798} C_VEL
LIN {X 0,Y 608.455,Z 984.998,A -85,B 0,C 180,E1 -457.799,E2 -457.799} C_VEL
LIN {X 0,Y 608.477,Z 974.61,A -85,B 0,C 180,E1 -458.802,E2 -458.802} C_VEL
LIN {X 0,Y 608.488,Z 963.763,A -85,B 0,C 180,E1 -459.64,E2 -459.64} C_VEL
LIN {X 0,Y 608.492,Z 952.793,A -85,B 0,C 180,E1 -460.312,E2 -460.312} C_VEL
LIN {X 0,Y 608.536,Z 940.792,A -85,B 0,C 180,E1 -460.889,E2 -460.889} C_VEL
LIN {X 0,Y 608.533,Z 928.913,A -85,B 0,C 180,E1 -461.322,E2 -461.322} C_VEL
LIN {X 0,Y 608.533,Z 916.57,A -85,B 0,C 180,E1 -461.638,E2 -461.638} C_VEL
LIN {X 0,Y 608.532,Z 900.825,A -85,B 0,C 180,E1 -461.87,E2 -461.87} C_VEL
LIN {X 0,Y 608.528,Z 801.939,A -85,B 0,C 180,E1 -463.057,E2 -463.057} C_VEL
LIN {X 0,Y 608.482,Z 776.958,A -85,B 0,C 180,E1 -465.576,E2 -465.576} C_VEL
LIN {X 0,Y 608.57,Z 751.743,A -85,B 0,C 180,E1 -468.167,E2 -468.167} C_VEL
LIN {X 0,Y 608.622,Z 724.847,A -85,B 0,C 180,E1 -470.974,E2 -470.974} C_VEL
LIN {X 0,Y 608.618,Z 699.632,A -85,B 0,C 180,E1 -473.657,E2 -473.657} C_VEL
LIN {X 0,Y 608.702,Z 677.779,A -85,B 0,C 180,E1 -476.022,E2 -476.022} C_VEL
LIN {X 0,Y 608.481,Z 676.744,A -85,B 0,C 180,E1 -476.194,E2 -476.194} C_VEL
LIN {X 0,Y 608.462,Z 676.686,A -85,B 0,C 180,E1 -479.019,E2 -479.019} C_VEL
LIN {X 0,Y 608.44,Z 676.688,A -85,B 0,C 180,E1 -481.317,E2 -481.317} C_VEL
LIN {X 0,Y 608.44,Z 676.69,A -85,B 0,C 180,E1 -483.73,E2 -483.73} C_VEL
LIN {X 0,Y 608.438,Z 676.693,A -85,B 0,C 180,E1 -486.091,E2 -486.091} C_VEL
LIN {X 0,Y 608.46,Z 676.696,A -85,B 0,C 180,E1 -488.587,E2 -488.587} C_VEL
LIN {X 0,Y 608.464,Z 676.686,A -85,B 0,C 180,E1 -491.342,E2 -491.342} C_VEL
LIN {X 0,Y 608.452,Z 676.687,A -85,B 0,C 180,E1 -493.869,E2 -493.869} C_VEL
LIN {X 0,Y 608.478,Z 676.692,A -85,B 0,C 180,E1 -496.688,E2 -496.688} C_VEL
LIN {X 0,Y 608.446,Z 676.687,A -85,B 0,C 180,E1 -499.696,E2 -499.696} C_VEL
LIN {X 0,Y 608.458,Z 676.686,A -85,B 0,C 180,E1 -502.253,E2 -502.253} C_VEL
LIN {X 0,Y 608.48,Z 676.694,A -85,B 0,C 180,E1 -505.088,E2 -505.088} C_VEL
LIN {X 0,Y 608.461,Z 676.686,A -85,B 0,C 180,E1 -507.905,E2 -507.905} C_VEL
LIN {X 0,Y 608.463,Z 676.685,A -85,B 0,C 180,E1 -510.22,E2 -510.22} C_VEL
LIN {X 0,Y 608.456,Z 676.688,A -85,B 0,C 180,E1 -512.794,E2 -512.794} C_VEL
LIN {X 0,Y 608.444,Z 676.698,A -85,B 0,C 180,E1 -515.429,E2 -515.429} C_VEL
LIN {X 0,Y 608.46,Z 676.686,A -85,B 0,C 180,E1 -518.308,E2 -518.308} C_VEL
LIN {X 0,Y 608.44,Z 676.69,A -85,B 0,C 180,E1 -521.13,E2 -521.13} C_VEL
LIN {X 0,Y 608.457,Z 676.695,A -85,B 0,C 180,E1 -523.906,E2 -523.906} C_VEL
LIN {X 0,Y 608.455,Z 676.686,A -85,B 0,C 180,E1 -526.643,E2 -526.643} C_VEL
LIN {X 0,Y 608.438,Z 676.69,A -85,B 0,C 180,E1 -529.35,E2 -529.35} C_VEL
LIN {X 0,Y 608.473,Z 676.695,A -85,B 0,C 180,E1 -532.033,E2 -532.033} C_VEL
LIN {X 0,Y 608.47,Z 676.687,A -85,B 0,C 180,E1 -534.698,E2 -534.698} C_VEL
LIN {X 0,Y 608.453,Z 676.686,A -85,B 0,C 180,E1 -537.352,E2 -537.352} C_VEL
LIN {X 0,Y 608.456,Z 676.691,A -85,B 0,C 180,E1 -540,E2 -540} C_VEL
LIN {X 0,Y 608.481,Z 676.691,A -85,B 0,C 180,E1 -542.648,E2 -542.648} C_VEL
LIN {X 0,Y 608.462,Z 676.686,A -85,B 0,C 180,E1 -545.302,E2 -545.302} C_VEL
LIN {X 0,Y 608.452,Z 676.687,A -85,B 0,C 180,E1 -547.967,E2 -547.967} C_VEL
LIN {X 0,Y 608.452,Z 676.687,A -85,B 0,C 180,E1 -549.47,E2 -549.47} C_VEL
LIN {X 0,Y 607.756,Z 676.775,A -85,B 0,C 180,E1 -550.023,E2 -550.023} C_VEL
LIN {X 0,Y 604.892,Z 677.138,A -85,B 0,C 180,E1 -550.92,E2 -550.92} C_VEL
LIN {X 0,Y 602.495,Z 677.432,A -85,B 0,C 180,E1 -551.641,E2 -551.641} C_VEL
LIN {X 0,Y 601.473,Z 677.558,A -85,B 0,C 180,E1 -552.198,E2 -552.198} C_VEL
LIN {X 0,Y 601.393,Z 677.57,A -85,B 0,C 180,E1 -552.386,E2 -552.386} C_VEL
LIN {X 0,Y 601.419,Z 677.574,A -85,B 0,C 180,E1 -554.897,E2 -554.897} C_VEL
LIN {X 0,Y 601.386,Z 677.568,A -85,B 0,C 180,E1 -557.689,E2 -557.689} C_VEL
LIN {X 0,Y 601.405,Z 677.566,A -85,B 0,C 180,E1 -560.523,E2 -560.523} C_VEL
LIN {X 0,Y 601.412,Z 677.57,A -85,B 0,C 180,E1 -563.411,E2 -563.411} C_VEL
LIN {X 0,Y 601.386,Z 677.567,A -85,B 0,C 180,E1 -566.365,E2 -566.365} C_VEL
LIN {X 0,Y 601.407,Z 677.565,A -85,B 0,C 180,E1 -568.786,E2 -568.786} C_VEL
LIN {X 0,Y 601.411,Z 677.575,A -85,B 0,C 180,E1 -571.456,E2 -571.456} C_VEL
LIN {X 0,Y 601.421,Z 677.565,A -85,B 0,C 180,E1 -574.119,E2 -574.119} C_VEL
LIN {X 0,Y 601.391,Z 677.566,A -85,B 0,C 180,E1 -576.584,E2 -576.584} C_VEL
LIN {X 0,Y 601.394,Z 677.567,A -85,B 0,C 180,E1 -579.128,E2 -579.128} C_VEL
LIN {X 0,Y 601.418,Z 677.573,A -85,B 0,C 180,E1 -581.766,E2 -581.766} C_VEL
LIN {X 0,Y 601.418,Z 677.565,A -85,B 0,C 180,E1 -584.536,E2 -584.536} C_VEL
LIN {X 0,Y 601.37,Z 677.57,A -85,B 0,C 180,E1 -587.328,E2 -587.328} C_VEL
LIN {X 0,Y 601.398,Z 677.575,A -85,B 0,C 180,E1 -590.006,E2 -590.006} C_VEL
LIN {X 0,Y 601.458,Z 677.722,A -85,B 0,C 180,E1 -592.056,E2 -592.056} C_VEL
LIN {X 0,Y 601.654,Z 678.725,A -85,B 0,C 180,E1 -592.163,E2 -592.163} C_VEL
LIN {X 0,Y 601.618,Z 762.718,A -85,B 0,C 180,E1 -593.199,E2 -593.199} C_VEL
LIN {X 0,Y 601.58,Z 775.789,A -85,B 0,C 180,E1 -593.499,E2 -593.499} C_VEL
LIN {X 0,Y 601.557,Z 787.572,A -85,B 0,C 180,E1 -593.896,E2 -593.896} C_VEL
LIN {X 0,Y 601.533,Z 799.398,A -85,B 0,C 180,E1 -594.429,E2 -594.429} C_VEL
LIN {X 0,Y 601.451,Z 810.474,A -85,B 0,C 180,E1 -595.072,E2 -595.072} C_VEL
LIN {X 0,Y 601.439,Z 821.596,A -85,B 0,C 180,E1 -595.884,E2 -595.884} C_VEL
LIN {X 0,Y 601.409,Z 830.433,A -85,B 0,C 180,E1 -596.687,E2 -596.687} C_VEL
LIN {X 0,Y 601.407,Z 837.906,A -85,B 0,C 180,E1 -597.484,E2 -597.484} C_VEL
LIN {X 0,Y 601.38,Z 845.952,A -85,B 0,C 180,E1 -598.552,E2 -598.552} C_VEL
LIN {X 0,Y 601.353,Z 852.46,A -85,B 0,C 180,E1 -599.639,E2 -599.639} C_VEL
LIN {X 0,Y 601.352,Z 857.017,A -85,B 0,C 180,E1 -600.605,E2 -600.605} C_VEL
LIN {X 0,Y 601.34,Z 861.132,A -85,B 0,C 180,E1 -601.751,E2 -601.751} C_VEL
LIN {X 0,Y 601.334,Z 863.933,A -85,B 0,C 180,E1 -602.885,E2 -602.885} C_VEL
LIN {X 0,Y 601.335,Z 865.627,A -85,B 0,C 180,E1 -604.149,E2 -604.149} C_VEL
LIN {X 0,Y 601.329,Z 865.989,A -85,B 0,C 180,E1 -605.119,E2 -605.119} C_VEL
LIN {X 0,Y 601.346,Z 865.685,A -85,B 0,C 180,E1 -605.856,E2 -605.856} C_VEL
LIN {X 0,Y 601.326,Z 864.946,A -85,B 0,C 180,E1 -606.587,E2 -606.587} C_VEL
LIN {X 0,Y 601.334,Z 863.486,A -85,B 0,C 180,E1 -607.415,E2 -607.415} C_VEL
LIN {X 0,Y 601.341,Z 860.941,A -85,B 0,C 180,E1 -608.4,E2 -608.4} C_VEL
LIN {X 0,Y 601.355,Z 857.054,A -85,B 0,C 180,E1 -609.477,E2 -609.477} C_VEL
LIN {X 0,Y 601.379,Z 851.943,A -85,B 0,C 180,E1 -610.546,E2 -610.546} C_VEL
LIN {X 0,Y 601.376,Z 845.484,A -85,B 0,C 180,E1 -611.608,E2 -611.608} C_VEL
LIN {X 0,Y 601.399,Z 837.397,A -85,B 0,C 180,E1 -612.664,E2 -612.664} C_VEL
LIN {X 0,Y 601.425,Z 828.512,A -85,B 0,C 180,E1 -613.594,E2 -613.594} C_VEL
LIN {X 0,Y 601.446,Z 819.034,A -85,B 0,C 180,E1 -614.411,E2 -614.411} C_VEL
LIN {X 0,Y 601.477,Z 807.706,A -85,B 0,C 180,E1 -615.192,E2 -615.192} C_VEL
LIN {X 0,Y 601.532,Z 796.599,A -85,B 0,C 180,E1 -615.798,E2 -615.798} C_VEL
LIN {X 0,Y 601.567,Z 785.214,A -85,B 0,C 180,E1 -616.284,E2 -616.284} C_VEL
LIN {X 0,Y 601.591,Z 772.482,A -85,B 0,C 180,E1 -616.683,E2 -616.683} C_VEL
LIN {X 0,Y 601.601,Z 759.647,A -85,B 0,C 180,E1 -616.941,E2 -616.941} C_VEL
LIN {X 0,Y 601.667,Z 678.681,A -85,B 0,C 180,E1 -617.928,E2 -617.928} C_VEL
LIN {X 0,Y 601.421,Z 677.672,A -85,B 0,C 180,E1 -618.051,E2 -618.051} C_VEL
LIN {X 0,Y 601.374,Z 677.57,A -85,B 0,C 180,E1 -620.584,E2 -620.584} C_VEL
LIN {X 0,Y 601.37,Z 677.571,A -85,B 0,C 180,E1 -622.615,E2 -622.615} C_VEL
LIN {X 0,Y 601.387,Z 677.569,A -85,B 0,C 180,E1 -624.637,E2 -624.637} C_VEL
LIN {X 0,Y 601.399,Z 677.566,A -85,B 0,C 180,E1 -627.322,E2 -627.322} C_VEL
LIN {X 0,Y 601.445,Z 677.566,A -85,B 0,C 180,E1 -630.001,E2 -630.001} C_VEL
LIN {X 0,Y 601.415,Z 677.568,A -85,B 0,C 180,E1 -632.68,E2 -632.68} C_VEL
LIN {X 0,Y 601.378,Z 677.568,A -85,B 0,C 180,E1 -635.365,E2 -635.365} C_VEL
LIN {X 0,Y 601.396,Z 677.569,A -85,B 0,C 180,E1 -638.062,E2 -638.062} C_VEL
LIN {X 0,Y 601.373,Z 677.572,A -85,B 0,C 180,E1 -640.984,E2 -640.984} C_VEL
LIN {X 0,Y 601.371,Z 677.569,A -85,B 0,C 180,E1 -643.518,E2 -643.518} C_VEL
LIN {X 0,Y 601.418,Z 677.566,A -85,B 0,C 180,E1 -646.288,E2 -646.288} C_VEL
LIN {X 0,Y 601.405,Z 677.57,A -85,B 0,C 180,E1 -649.1,E2 -649.1} C_VEL
LIN {X 0,Y 601.387,Z 677.572,A -85,B 0,C 180,E1 -651.241,E2 -651.241} C_VEL
LIN {X 0,Y 601.365,Z 677.573,A -85,B 0,C 180,E1 -653.413,E2 -653.413} C_VEL
LIN {X 0,Y 601.353,Z 677.57,A -85,B 0,C 180,E1 -655.855,E2 -655.855} C_VEL
LIN {X 0,Y 601.351,Z 677.571,A -85,B 0,C 180,E1 -657.872,E2 -657.872} C_VEL
LIN {X 0,Y 601.348,Z 677.571,A -85,B 0,C 180,E1 -660.169,E2 -660.169} C_VEL
LIN {X 0,Y 601.388,Z 677.569,A -85,B 0,C 180,E1 -662.71,E2 -662.71} C_VEL
LIN {X 0,Y 601.349,Z 677.575,A -85,B 0,C 180,E1 -665.758,E2 -665.758} C_VEL
LIN {X 0,Y 601.341,Z 677.572,A -85,B 0,C 180,E1 -668.275,E2 -668.275} C_VEL
LIN {X 0,Y 601.37,Z 677.57,A -85,B 0,C 180,E1 -670.879,E2 -670.879} C_VEL
LIN {X 0,Y 601.409,Z 677.576,A -85,B 0,C 180,E1 -673.589,E2 -673.589} C_VEL
LIN {X 0,Y 601.379,Z 677.568,A -85,B 0,C 180,E1 -676.433,E2 -676.433} C_VEL
LIN {X 0,Y 601.351,Z 677.573,A -85,B 0,C 180,E1 -679.12,E2 -679.12} C_VEL
LIN {X 0,Y 601.381,Z 677.577,A -85,B 0,C 180,E1 -681.729,E2 -681.729} C_VEL
LIN {X 0,Y 601.37,Z 677.574,A -85,B 0,C 180,E1 -684.244,E2 -684.244} C_VEL
LIN {X 0,Y 601.363,Z 677.571,A -85,B 0,C 180,E1 -686.682,E2 -686.682} C_VEL
LIN {X 0,Y 601.362,Z 677.57,A -85,B 0,C 180,E1 -689.054,E2 -689.054} C_VEL
LIN {X 0,Y 601.353,Z 677.572,A -85,B 0,C 180,E1 -691.369,E2 -691.369} C_VEL
LIN {X 0,Y 601.469,Z 677.742,A -85,B 0,C 180,E1 -694.061,E2 -694.061} C_VEL
LIN {X 0,Y 601.676,Z 678.97,A -85,B 0,C 180,E1 -694.173,E2 -694.173} C_VEL
LIN {X 0,Y 601.587,Z 762.213,A -85,B 0,C 180,E1 -695.19,E2 -695.19} C_VEL
LIN {X 0,Y 601.594,Z 775.473,A -85,B 0,C 180,E1 -695.491,E2 -695.491} C_VEL
LIN {X 0,Y 601.565,Z 787.902,A -85,B 0,C 180,E1 -695.91,E2 -695.91} C_VEL
LIN {X 0,Y 601.514,Z 799.031,A -85,B 0,C 180,E1 -696.411,E2 -696.411} C_VEL
LIN {X 0,Y 601.471,Z 810.091,A -85,B 0,C 180,E1 -697.047,E2 -697.047} C_VEL
LIN {X 0,Y 601.465,Z 821.349,A -85,B 0,C 180,E1 -697.864,E2 -697.864} C_VEL
LIN {X 0,Y 601.414,Z 829.355,A -85,B 0,C 180,E1 -698.581,E2 -698.581} C_VEL
LIN {X 0,Y 601.385,Z 837.836,A -85,B 0,C 180,E1 -699.476,E2 -699.476} C_VEL
LIN {X 0,Y 601.386,Z 845.897,A -85,B 0,C 180,E1 -700.545,E2 -700.545} C_VEL
LIN {X 0,Y 601.351,Z 852.275,A -85,B 0,C 180,E1 -701.606,E2 -701.606} C_VEL
LIN {X 0,Y 601.341,Z 857.253,A -85,B 0,C 180,E1 -702.661,E2 -702.661} C_VEL
LIN {X 0,Y 601.349,Z 861.003,A -85,B 0,C 180,E1 -703.71,E2 -703.71} C_VEL
LIN {X 0,Y 601.326,Z 862.897,A -85,B 0,C 180,E1 -704.406,E2 -704.406} C_VEL
LIN {X 0,Y 601.315,Z 864.307,A -85,B 0,C 180,E1 -705.1,E2 -705.1} C_VEL
LIN {X 0,Y 601.354,Z 865.452,A -85,B 0,C 180,E1 -705.936,E2 -705.936} C_VEL
LIN {X 0,Y 601.324,Z 865.977,A -85,B 0,C 180,E1 -707.17,E2 -707.17} C_VEL
LIN {X 0,Y 601.342,Z 865.685,A -85,B 0,C 180,E1 -707.856,E2 -707.856} C_VEL
LIN {X 0,Y 601.343,Z 864.239,A -85,B 0,C 180,E1 -709.032,E2 -709.032} C_VEL
LIN {X 0,Y 601.328,Z 862.34,A -85,B 0,C 180,E1 -709.903,E2 -709.903} C_VEL
LIN {X 0,Y 601.348,Z 859.207,A -85,B 0,C 180,E1 -710.922,E2 -710.922} C_VEL
LIN {X 0,Y 601.35,Z 855.019,A -85,B 0,C 180,E1 -711.938,E2 -711.938} C_VEL
LIN {X 0,Y 601.384,Z 848.642,A -85,B 0,C 180,E1 -713.12,E2 -713.12} C_VEL
LIN {X 0,Y 601.386,Z 841.724,A -85,B 0,C 180,E1 -714.131,E2 -714.131} C_VEL
LIN {X 0,Y 601.419,Z 834.682,A -85,B 0,C 180,E1 -714.972,E2 -714.972} C_VEL
LIN {X 0,Y 601.421,Z 824.279,A -85,B 0,C 180,E1 -715.979,E2 -715.979} C_VEL
LIN {X 0,Y 601.485,Z 813.466,A -85,B 0,C 180,E1 -716.818,E2 -716.818} C_VEL
LIN {X 0,Y 601.51,Z 802.599,A -85,B 0,C 180,E1 -717.489,E2 -717.489} C_VEL
LIN {X 0,Y 601.536,Z 789.538,A -85,B 0,C 180,E1 -718.117,E2 -718.117} C_VEL
LIN {X 0,Y 601.603,Z 776.966,A -85,B 0,C 180,E1 -718.556,E2 -718.556} C_VEL
LIN {X 0,Y 601.594,Z 763.814,A -85,B 0,C 180,E1 -718.87,E2 -718.87} C_VEL
LIN {X 0,Y 601.64,Z 739.893,A -85,B 0,C 180,E1 -719.184,E2 -719.184} C_VEL
LIN {X 0,Y 601.675,Z 679.134,A -85,B 0,C 180,E1 -719.916,E2 -719.916} C_VEL
LIN {X 0,Y 601.47,Z 677.889,A -85,B 0,C 180,E1 -720,E2 -720} C_VEL
LIN {X 0,Y 601.433,Z 677.565,A -85,B 0,C 180,E1 -720.335,E2 -720.335} C_VEL
LIN {X 0,Y 601.431,Z 677.563,A -85,B 0,C 180,E1 -722.679,E2 -722.679} C_VEL
LIN {X 0,Y 601.432,Z 677.563,A -85,B 0,C 180,E1 -725.364,E2 -725.364} C_VEL
LIN {X 0,Y 601.439,Z 677.571,A -85,B 0,C 180,E1 -728.061,E2 -728.061} C_VEL
LIN {X 0,Y 601.421,Z 677.563,A -85,B 0,C 180,E1 -731.007,E2 -731.007} C_VEL
LIN {X 0,Y 601.412,Z 677.564,A -85,B 0,C 180,E1 -733.516,E2 -733.516} C_VEL
LIN {X 0,Y 601.442,Z 677.57,A -85,B 0,C 180,E1 -736.287,E2 -736.287} C_VEL
LIN {X 0,Y 601.418,Z 677.565,A -85,B 0,C 180,E1 -739.099,E2 -739.099} C_VEL
LIN {X 0,Y 601.403,Z 677.566,A -85,B 0,C 180,E1 -741.239,E2 -741.239} C_VEL
LIN {X 0,Y 601.456,Z 677.561,A -85,B 0,C 180,E1 -744.14,E2 -744.14} C_VEL
LIN {X 0,Y 601.407,Z 677.569,A -85,B 0,C 180,E1 -747.113,E2 -747.113} C_VEL
LIN {X 0,Y 601.416,Z 677.565,A -85,B 0,C 180,E1 -749.393,E2 -749.393} C_VEL
LIN {X 0,Y 601.402,Z 677.565,A -85,B 0,C 180,E1 -751.727,E2 -751.727} C_VEL
LIN {X 0,Y 601.424,Z 677.562,A -85,B 0,C 180,E1 -754.119,E2 -754.119} C_VEL
LIN {X 0,Y 601.439,Z 677.566,A -85,B 0,C 180,E1 -757.381,E2 -757.381} C_VEL
LIN {X 0,Y 601.405,Z 677.565,A -85,B 0,C 180,E1 -759.996,E2 -759.996} C_VEL
LIN {X 0,Y 601.417,Z 677.565,A -85,B 0,C 180,E1 -762.67,E2 -762.67} C_VEL
LIN {X 0,Y 601.405,Z 677.573,A -85,B 0,C 180,E1 -765.479,E2 -765.479} C_VEL
LIN {X 0,Y 601.423,Z 677.562,A -85,B 0,C 180,E1 -768.407,E2 -768.407} C_VEL
LIN {X 0,Y 601.404,Z 677.566,A -85,B 0,C 180,E1 -770.872,E2 -770.872} C_VEL
LIN {X 0,Y 601.404,Z 677.573,A -85,B 0,C 180,E1 -773.416,E2 -773.416} C_VEL
LIN {X 0,Y 601.421,Z 677.567,A -85,B 0,C 180,E1 -776.066,E2 -776.066} C_VEL
LIN {X 0,Y 601.421,Z 677.563,A -85,B 0,C 180,E1 -778.546,E2 -778.546} C_VEL
LIN {X 0,Y 601.431,Z 677.565,A -85,B 0,C 180,E1 -781.372,E2 -781.372} C_VEL
LIN {X 0,Y 601.445,Z 677.785,A -85,B 0,C 180,E1 -783.626,E2 -783.626} C_VEL
LIN {X 0,Y 601.98,Z 681.003,A -85,B 0,C 180,E1 -784.022,E2 -784.022} C_VEL
LIN {X 0,Y 601.808,Z 704.655,A -85,B 0,C 180,E1 -786.605,E2 -786.605} C_VEL
LIN {X 0,Y 601.742,Z 731.551,A -85,B 0,C 180,E1 -789.488,E2 -789.488} C_VEL
LIN {X 0,Y 601.622,Z 758.447,A -85,B 0,C 180,E1 -792.318,E2 -792.318} C_VEL
LIN {X 0,Y 601.525,Z 785.343,A -85,B 0,C 180,E1 -795.105,E2 -795.105} C_VEL
LIN {X 0,Y 601.514,Z 801.904,A -85,B 0,C 180,E1 -796.786,E2 -796.786} C_VEL
LIN {X 0,Y 601.697,Z 809.431,A -85,B 0,C 180,E1 -796.898,E2 -796.898} C_VEL
LIN {X 0,Y 601.601,Z 911.896,A -85,B 0,C 180,E1 -798.138,E2 -798.138} C_VEL
LIN {X 0,Y 601.587,Z 925.183,A -85,B 0,C 180,E1 -798.437,E2 -798.437} C_VEL
LIN {X 0,Y 601.55,Z 936.906,A -85,B 0,C 180,E1 -798.826,E2 -798.826} C_VEL
LIN {X 0,Y 601.531,Z 947.903,A -85,B 0,C 180,E1 -799.31,E2 -799.31} C_VEL
LIN {X 0,Y 601.462,Z 958.564,A -85,B 0,C 180,E1 -799.905,E2 -799.905} C_VEL
LIN {X 0,Y 601.447,Z 969.463,A -85,B 0,C 180,E1 -800.668,E2 -800.668} C_VEL
LIN {X 0,Y 601.423,Z 978.301,A -85,B 0,C 180,E1 -801.431,E2 -801.431} C_VEL
LIN {X 0,Y 601.418,Z 987.952,A -85,B 0,C 180,E1 -802.445,E2 -802.445} C_VEL
LIN {X 0,Y 601.366,Z 995.244,A -85,B 0,C 180,E1 -803.401,E2 -803.401} C_VEL
LIN {X 0,Y 601.372,Z 1000.861,A -85,B 0,C 180,E1 -804.298,E2 -804.298} C_VEL
LIN {X 0,Y 601.336,Z 1005.946,A -85,B 0,C 180,E1 -805.306,E2 -805.306} C_VEL
LIN {X 0,Y 601.367,Z 1009.893,A -85,B 0,C 180,E1 -806.314,E2 -806.314} C_VEL
LIN {X 0,Y 601.325,Z 1012.807,A -85,B 0,C 180,E1 -807.319,E2 -807.319} C_VEL
LIN {X 0,Y 601.341,Z 1014.2,A -85,B 0,C 180,E1 -807.99,E2 -807.99} C_VEL
LIN {X 0,Y 601.339,Z 1015.783,A -85,B 0,C 180,E1 -809.329,E2 -809.329} C_VEL
LIN {X 0,Y 601.335,Z 1016,A -85,B 0,C 180,E1 -809.999,E2 -809.999} C_VEL
LIN {X 0,Y 601.347,Z 1015.185,A -85,B 0,C 180,E1 -811.338,E2 -811.338} C_VEL
LIN {X 0,Y 601.341,Z 1014.203,A -85,B 0,C 180,E1 -812.008,E2 -812.008} C_VEL
LIN {X 0,Y 601.325,Z 1012.812,A -85,B 0,C 180,E1 -812.679,E2 -812.679} C_VEL
LIN {X 0,Y 601.367,Z 1009.899,A -85,B 0,C 180,E1 -813.684,E2 -813.684} C_VEL
LIN {X 0,Y 601.336,Z 1005.954,A -85,B 0,C 180,E1 -814.692,E2 -814.692} C_VEL
LIN {X 0,Y 601.372,Z 999.883,A -85,B 0,C 180,E1 -815.868,E2 -815.868} C_VEL
LIN {X 0,Y 601.38,Z 993.243,A -85,B 0,C 180,E1 -816.879,E2 -816.879} C_VEL
LIN {X 0,Y 601.4,Z 984.999,A -85,B 0,C 180,E1 -817.891,E2 -817.891} C_VEL
LIN {X 0,Y 601.434,Z 974.611,A -85,B 0,C 180,E1 -818.906,E2 -818.906} C_VEL
LIN {X 0,Y 601.46,Z 963.763,A -85,B 0,C 180,E1 -819.754,E2 -819.754} C_VEL
LIN {X 0,Y 601.495,Z 952.794,A -85,B 0,C 180,E1 -820.433,E2 -820.433} C_VEL
LIN {X 0,Y 601.55,Z 940.657,A -85,B 0,C 180,E1 -821.023,E2 -821.023} C_VEL
LIN {X 0,Y 601.578,Z 928.912,A -85,B 0,C 180,E1 -821.454,E2 -821.454} C_VEL
LIN {X 0,Y 601.587,Z 916.569,A -85,B 0,C 180,E1 -821.774,E2 -821.774} C_VEL
LIN {X 0,Y 601.601,Z 900.825,A -85,B 0,C 180,E1 -822.009,E2 -822.009} C_VEL
LIN {X 0,Y 601.572,Z 802.61,A -85,B 0,C 180,E1 -823.189,E2 -823.189} C_VEL
LIN {X 0,Y 601.512,Z 801.432,A -85,B 0,C 180,E1 -823.255,E2 -823.255} C_VEL
LIN {X 0,Y 601.529,Z 775.277,A -85,B 0,C 180,E1 -825.935,E2 -825.935} C_VEL
LIN {X 0,Y 601.674,Z 748.142,A -85,B 0,C 180,E1 -828.761,E2 -828.761} C_VEL
LIN {X 0,Y 601.755,Z 723.166,A -85,B 0,C 180,E1 -831.405,E2 -831.405} C_VEL
LIN {X 0,Y 601.807,Z 699.632,A -85,B 0,C 180,E1 -833.941,E2 -833.941} C_VEL
LIN {X 0,Y 601.962,Z 680.005,A -85,B 0,C 180,E1 -836.089,E2 -836.089} C_VEL
LIN {X 0,Y 601.424,Z 677.634,A -85,B 0,C 180,E1 -836.42,E2 -836.42} C_VEL
LIN {X 0,Y 601.435,Z 677.563,A -85,B 0,C 180,E1 -838.788,E2 -838.788} C_VEL
LIN {X 0,Y 601.415,Z 677.564,A -85,B 0,C 180,E1 -841.453,E2 -841.453} C_VEL
LIN {X 0,Y 601.415,Z 677.57,A -85,B 0,C 180,E1 -844.118,E2 -844.118} C_VEL
LIN {X 0,Y 601.431,Z 677.561,A -85,B 0,C 180,E1 -847.381,E2 -847.381} C_VEL
LIN {X 0,Y 601.395,Z 677.568,A -85,B 0,C 180,E1 -849.995,E2 -849.995} C_VEL
LIN {X 0,Y 601.404,Z 677.576,A -85,B 0,C 180,E1 -852.669,E2 -852.669} C_VEL
LIN {X 0,Y 601.418,Z 677.563,A -85,B 0,C 180,E1 -855.481,E2 -855.481} C_VEL
LIN {X 0,Y 601.414,Z 677.567,A -85,B 0,C 180,E1 -858.406,E2 -858.406} C_VEL
LIN {X 0,Y 601.431,Z 677.571,A -85,B 0,C 180,E1 -860.875,E2 -860.875} C_VEL
LIN {X 0,Y 601.436,Z 677.561,A -85,B 0,C 180,E1 -863.733,E2 -863.733} C_VEL
LIN {X 0,Y 601.424,Z 677.562,A -85,B 0,C 180,E1 -866.063,E2 -866.063} C_VEL
LIN {X 0,Y 601.408,Z 677.565,A -85,B 0,C 180,E1 -868.545,E2 -868.545} C_VEL
LIN {X 0,Y 601.434,Z 677.57,A -85,B 0,C 180,E1 -871.209,E2 -871.209} C_VEL
LIN {X 0,Y 601.397,Z 677.573,A -85,B 0,C 180,E1 -873.636,E2 -873.636} C_VEL
LIN {X 0,Y 601.408,Z 677.564,A -85,B 0,C 180,E1 -876.589,E2 -876.589} C_VEL
LIN {X 0,Y 601.423,Z 677.57,A -85,B 0,C 180,E1 -879.478,E2 -879.478} C_VEL
LIN {X 0,Y 601.387,Z 677.568,A -85,B 0,C 180,E1 -882.311,E2 -882.311} C_VEL
LIN {X 0,Y 601.406,Z 677.566,A -85,B 0,C 180,E1 -884.409,E2 -884.409} C_VEL
LIN {X 0,Y 601.402,Z 677.565,A -85,B 0,C 180,E1 -887.171,E2 -887.171} C_VEL
LIN {X 0,Y 601.427,Z 677.571,A -85,B 0,C 180,E1 -889.905,E2 -889.905} C_VEL
LIN {X 0,Y 601.446,Z 677.562,A -85,B 0,C 180,E1 -892.615,E2 -892.615} C_VEL
LIN {X 0,Y 601.399,Z 677.565,A -85,B 0,C 180,E1 -895.308,E2 -895.308} C_VEL
LIN {X 0,Y 601.408,Z 677.57,A -85,B 0,C 180,E1 -897.991,E2 -897.991} C_VEL
LIN {X 0,Y 601.451,Z 677.565,A -85,B 0,C 180,E1 -900.67,E2 -900.67} C_VEL
LIN {X 0,Y 601.422,Z 677.562,A -85,B 0,C 180,E1 -903.35,E2 -903.35} C_VEL
LIN {X 0,Y 601.386,Z 677.569,A -85,B 0,C 180,E1 -906.038,E2 -906.038} C_VEL
LIN {X 0,Y 601.434,Z 677.571,A -85,B 0,C 180,E1 -908.738,E2 -908.738} C_VEL
LIN {X 0,Y 601.425,Z 677.563,A -85,B 0,C 180,E1 -911.458,E2 -911.458} C_VEL
LIN {X 0,Y 601.393,Z 677.57,A -85,B 0,C 180,E1 -912.386,E2 -912.386} C_VEL
LIN {X 0,Y 600.735,Z 677.659,A -85,B 0,C 180,E1 -912.946,E2 -912.946} C_VEL
LIN {X 0,Y 597.888,Z 678.017,A -85,B 0,C 180,E1 -913.854,E2 -913.854} C_VEL
LIN {X 0,Y 595.475,Z 678.314,A -85,B 0,C 180,E1 -914.584,E2 -914.584} C_VEL
LIN {X 0,Y 594.435,Z 678.439,A -85,B 0,C 180,E1 -915.147,E2 -915.147} C_VEL
LIN {X 0,Y 594.349,Z 678.447,A -85,B 0,C 180,E1 -915.338,E2 -915.338} C_VEL
LIN {X 0,Y 594.335,Z 678.445,A -85,B 0,C 180,E1 -917.906,E2 -917.906} C_VEL
LIN {X 0,Y 594.382,Z 678.445,A -85,B 0,C 180,E1 -920.777,E2 -920.777} C_VEL
LIN {X 0,Y 594.369,Z 678.443,A -85,B 0,C 180,E1 -923.705,E2 -923.705} C_VEL
LIN {X 0,Y 594.359,Z 678.443,A -85,B 0,C 180,E1 -926.02,E2 -926.02} C_VEL
LIN {X 0,Y 594.357,Z 678.442,A -85,B 0,C 180,E1 -928.228,E2 -928.228} C_VEL
LIN {X 0,Y 594.369,Z 678.441,A -85,B 0,C 180,E1 -930.561,E2 -930.561} C_VEL
LIN {X 0,Y 594.368,Z 678.443,A -85,B 0,C 180,E1 -932.951,E2 -932.951} C_VEL
LIN {X 0,Y 594.346,Z 678.451,A -85,B 0,C 180,E1 -935.41,E2 -935.41} C_VEL
LIN {X 0,Y 594.381,Z 678.446,A -85,B 0,C 180,E1 -937.942,E2 -937.942} C_VEL
LIN {X 0,Y 594.36,Z 678.442,A -85,B 0,C 180,E1 -940.822,E2 -940.822} C_VEL
LIN {X 0,Y 594.358,Z 678.444,A -85,B 0,C 180,E1 -943.301,E2 -943.301} C_VEL
LIN {X 0,Y 594.355,Z 678.451,A -85,B 0,C 180,E1 -946.162,E2 -946.162} C_VEL
LIN {X 0,Y 594.364,Z 678.442,A -85,B 0,C 180,E1 -949.18,E2 -949.18} C_VEL
LIN {X 0,Y 594.429,Z 678.632,A -85,B 0,C 180,E1 -951.919,E2 -951.919} C_VEL
LIN {X 0,Y 594.699,Z 679.901,A -85,B 0,C 180,E1 -952.031,E2 -952.031} C_VEL
LIN {X 0,Y 594.675,Z 762.466,A -85,B 0,C 180,E1 -953.054,E2 -953.054} C_VEL
LIN {X 0,Y 594.625,Z 775.859,A -85,B 0,C 180,E1 -953.364,E2 -953.364} C_VEL
LIN {X 0,Y 594.575,Z 787.825,A -85,B 0,C 180,E1 -953.773,E2 -953.773} C_VEL
LIN {X 0,Y 594.525,Z 799.207,A -85,B 0,C 180,E1 -954.292,E2 -954.292} C_VEL
LIN {X 0,Y 594.473,Z 809.847,A -85,B 0,C 180,E1 -954.912,E2 -954.912} C_VEL
LIN {X 0,Y 594.421,Z 820.339,A -85,B 0,C 180,E1 -955.673,E2 -955.673} C_VEL
LIN {X 0,Y 594.38,Z 829.026,A -85,B 0,C 180,E1 -956.444,E2 -956.444} C_VEL
LIN {X 0,Y 594.355,Z 838.387,A -85,B 0,C 180,E1 -957.453,E2 -957.453} C_VEL
LIN {X 0,Y 594.323,Z 845.241,A -85,B 0,C 180,E1 -958.367,E2 -958.367} C_VEL
LIN {X 0,Y 594.287,Z 851.723,A -85,B 0,C 180,E1 -959.436,E2 -959.436} C_VEL
LIN {X 0,Y 594.275,Z 857.258,A -85,B 0,C 180,E1 -960.609,E2 -960.609} C_VEL
LIN {X 0,Y 594.242,Z 861.308,A -85,B 0,C 180,E1 -961.767,E2 -961.767} C_VEL
LIN {X 0,Y 594.26,Z 863.25,A -85,B 0,C 180,E1 -962.535,E2 -962.535} C_VEL
LIN {X 0,Y 594.225,Z 864.661,A -85,B 0,C 180,E1 -963.294,E2 -963.294} C_VEL
LIN {X 0,Y 594.228,Z 865.565,A -85,B 0,C 180,E1 -964.05,E2 -964.05} C_VEL
LIN {X 0,Y 594.219,Z 865.95,A -85,B 0,C 180,E1 -964.801,E2 -964.801} C_VEL
LIN {X 0,Y 594.236,Z 865.866,A -85,B 0,C 180,E1 -965.6,E2 -965.6} C_VEL
LIN {X 0,Y 594.224,Z 865.311,A -85,B 0,C 180,E1 -966.29,E2 -966.29} C_VEL
LIN {X 0,Y 594.244,Z 863.801,A -85,B 0,C 180,E1 -967.294,E2 -967.294} C_VEL
LIN {X 0,Y 594.247,Z 860.776,A -85,B 0,C 180,E1 -968.493,E2 -968.493} C_VEL
LIN {X 0,Y 594.284,Z 856.83,A -85,B 0,C 180,E1 -969.583,E2 -969.583} C_VEL
LIN {X 0,Y 594.297,Z 851.664,A -85,B 0,C 180,E1 -970.664,E2 -970.664} C_VEL
LIN {X 0,Y 594.32,Z 845.139,A -85,B 0,C 180,E1 -971.739,E2 -971.739} C_VEL
LIN {X 0,Y 594.327,Z 836.954,A -85,B 0,C 180,E1 -972.806,E2 -972.806} C_VEL
LIN {X 0,Y 594.394,Z 826.738,A -85,B 0,C 180,E1 -973.869,E2 -973.869} C_VEL
LIN {X 0,Y 594.416,Z 816.038,A -85,B 0,C 180,E1 -974.749,E2 -974.749} C_VEL
LIN {X 0,Y 594.477,Z 805.429,A -85,B 0,C 180,E1 -975.451,E2 -975.451} C_VEL
LIN {X 0,Y 594.56,Z 793.35,A -85,B 0,C 180,E1 -976.081,E2 -976.081} C_VEL
LIN {X 0,Y 594.596,Z 780.331,A -85,B 0,C 180,E1 -976.588,E2 -976.588} C_VEL
LIN {X 0,Y 594.668,Z 767.523,A -85,B 0,C 180,E1 -976.938,E2 -976.938} C_VEL
LIN {X 0,Y 594.687,Z 754.174,A -85,B 0,C 180,E1 -977.155,E2 -977.155} C_VEL
LIN {X 0,Y 594.718,Z 679.963,A -85,B 0,C 180,E1 -978.057,E2 -978.057} C_VEL
LIN {X 0,Y 594.423,Z 678.727,A -85,B 0,C 180,E1 -978.153,E2 -978.153} C_VEL
LIN {X 0,Y 594.374,Z 678.447,A -85,B 0,C 180,E1 -978.405,E2 -978.405} C_VEL
LIN {X 0,Y 594.357,Z 678.444,A -85,B 0,C 180,E1 -981.159,E2 -981.159} C_VEL
LIN {X 0,Y 594.36,Z 678.451,A -85,B 0,C 180,E1 -983.892,E2 -983.892} C_VEL
LIN {X 0,Y 594.316,Z 678.451,A -85,B 0,C 180,E1 -986.611,E2 -986.611} C_VEL
LIN {X 0,Y 594.343,Z 678.448,A -85,B 0,C 180,E1 -988.646,E2 -988.646} C_VEL
LIN {X 0,Y 594.333,Z 678.45,A -85,B 0,C 180,E1 -990.679,E2 -990.679} C_VEL
LIN {X 0,Y 594.38,Z 678.444,A -85,B 0,C 180,E1 -992.712,E2 -992.712} C_VEL
LIN {X 0,Y 594.347,Z 678.444,A -85,B 0,C 180,E1 -995.429,E2 -995.429} C_VEL
LIN {X 0,Y 594.351,Z 678.448,A -85,B 0,C 180,E1 -998.159,E2 -998.159} C_VEL
LIN {X 0,Y 594.336,Z 678.448,A -85,B 0,C 180,E1 -1001.045,E2 -1001.045} C_VEL
LIN {X 0,Y 594.34,Z 678.444,A -85,B 0,C 180,E1 -1003.681,E2 -1003.681} C_VEL
LIN {X 0,Y 594.389,Z 678.444,A -85,B 0,C 180,E1 -1006.486,E2 -1006.486} C_VEL
LIN {X 0,Y 594.352,Z 678.445,A -85,B 0,C 180,E1 -1009.336,E2 -1009.336} C_VEL
LIN {X 0,Y 594.342,Z 678.446,A -85,B 0,C 180,E1 -1011.505,E2 -1011.505} C_VEL
LIN {X 0,Y 594.332,Z 678.446,A -85,B 0,C 180,E1 -1013.707,E2 -1013.707} C_VEL
LIN {X 0,Y 594.358,Z 678.446,A -85,B 0,C 180,E1 -1016.702,E2 -1016.702} C_VEL
LIN {X 0,Y 594.318,Z 678.449,A -85,B 0,C 180,E1 -1019.78,E2 -1019.78} C_VEL
LIN {X 0,Y 594.336,Z 678.445,A -85,B 0,C 180,E1 -1022.15,E2 -1022.15} C_VEL
LIN {X 0,Y 594.324,Z 678.446,A -85,B 0,C 180,E1 -1024.585,E2 -1024.585} C_VEL
LIN {X 0,Y 594.357,Z 678.45,A -85,B 0,C 180,E1 -1027.604,E2 -1027.604} C_VEL
LIN {X 0,Y 594.318,Z 678.447,A -85,B 0,C 180,E1 -1030.572,E2 -1030.572} C_VEL
LIN {X 0,Y 594.311,Z 678.449,A -85,B 0,C 180,E1 -1032.846,E2 -1032.846} C_VEL
LIN {X 0,Y 594.313,Z 678.452,A -85,B 0,C 180,E1 -1035.197,E2 -1035.197} C_VEL
LIN {X 0,Y 594.35,Z 678.447,A -85,B 0,C 180,E1 -1038.156,E2 -1038.156} C_VEL
LIN {X 0,Y 594.325,Z 678.448,A -85,B 0,C 180,E1 -1041.19,E2 -1041.19} C_VEL
LIN {X 0,Y 594.341,Z 678.453,A -85,B 0,C 180,E1 -1043.754,E2 -1043.754} C_VEL
LIN {X 0,Y 594.342,Z 678.451,A -85,B 0,C 180,E1 -1046.236,E2 -1046.236} C_VEL
LIN {X 0,Y 594.314,Z 678.45,A -85,B 0,C 180,E1 -1048.646,E2 -1048.646} C_VEL
LIN {X 0,Y 594.333,Z 678.446,A -85,B 0,C 180,E1 -1051.052,E2 -1051.052} C_VEL
LIN {X 0,Y 594.416,Z 678.662,A -85,B 0,C 180,E1 -1053.925,E2 -1053.925} C_VEL
LIN {X 0,Y 594.655,Z 679.65,A -85,B 0,C 180,E1 -1054.023,E2 -1054.023} C_VEL
LIN {X 0,Y 594.638,Z 762.232,A -85,B 0,C 180,E1 -1055.05,E2 -1055.05} C_VEL
LIN {X 0,Y 594.636,Z 774.755,A -85,B 0,C 180,E1 -1055.334,E2 -1055.334} C_VEL
LIN {X 0,Y 594.561,Z 787.11,A -85,B 0,C 180,E1 -1055.747,E2 -1055.747} C_VEL
LIN {X 0,Y 594.512,Z 799.36,A -85,B 0,C 180,E1 -1056.301,E2 -1056.301} C_VEL
LIN {X 0,Y 594.446,Z 811.706,A -85,B 0,C 180,E1 -1057.036,E2 -1057.036} C_VEL
LIN {X 0,Y 594.423,Z 822.619,A -85,B 0,C 180,E1 -1057.86,E2 -1057.86} C_VEL
LIN {X 0,Y 594.36,Z 831.194,A -85,B 0,C 180,E1 -1058.665,E2 -1058.665} C_VEL
LIN {X 0,Y 594.332,Z 837.964,A -85,B 0,C 180,E1 -1059.403,E2 -1059.403} C_VEL
LIN {X 0,Y 594.307,Z 846.001,A -85,B 0,C 180,E1 -1060.484,E2 -1060.484} C_VEL
LIN {X 0,Y 594.289,Z 851.411,A -85,B 0,C 180,E1 -1061.379,E2 -1061.379} C_VEL
LIN {X 0,Y 594.262,Z 856.579,A -85,B 0,C 180,E1 -1062.448,E2 -1062.448} C_VEL
LIN {X 0,Y 594.248,Z 860.504,A -85,B 0,C 180,E1 -1063.51,E2 -1063.51} C_VEL
LIN {X 0,Y 594.253,Z 862.505,A -85,B 0,C 180,E1 -1064.216,E2 -1064.216} C_VEL
LIN {X 0,Y 594.21,Z 864.045,A -85,B 0,C 180,E1 -1064.918,E2 -1064.918} C_VEL
LIN {X 0,Y 594.266,Z 865.398,A -85,B 0,C 180,E1 -1065.876,E2 -1065.876} C_VEL
LIN {X 0,Y 594.243,Z 865.998,A -85,B 0,C 180,E1 -1067.014,E2 -1067.014} C_VEL
LIN {X 0,Y 594.24,Z 865.793,A -85,B 0,C 180,E1 -1067.708,E2 -1067.708} C_VEL
LIN {X 0,Y 594.244,Z 864.179,A -85,B 0,C 180,E1 -1069.092,E2 -1069.092} C_VEL
LIN {X 0,Y 594.231,Z 862.736,A -85,B 0,C 180,E1 -1069.781,E2 -1069.781} C_VEL
LIN {X 0,Y 594.264,Z 859.751,A -85,B 0,C 180,E1 -1070.813,E2 -1070.813} C_VEL
LIN {X 0,Y 594.28,Z 855.726,A -85,B 0,C 180,E1 -1071.841,E2 -1071.841} C_VEL
LIN {X 0,Y 594.307,Z 849.563,A -85,B 0,C 180,E1 -1073.038,E2 -1073.038} C_VEL
LIN {X 0,Y 594.319,Z 841.606,A -85,B 0,C 180,E1 -1074.231,E2 -1074.231} C_VEL
LIN {X 0,Y 594.358,Z 834.542,A -85,B 0,C 180,E1 -1075.082,E2 -1075.082} C_VEL
LIN {X 0,Y 594.405,Z 824.094,A -85,B 0,C 180,E1 -1076.102,E2 -1076.102} C_VEL
LIN {X 0,Y 594.443,Z 814.423,A -85,B 0,C 180,E1 -1076.865,E2 -1076.865} C_VEL
LIN {X 0,Y 594.505,Z 803.852,A -85,B 0,C 180,E1 -1077.544,E2 -1077.544} C_VEL
LIN {X 0,Y 594.547,Z 792.095,A -85,B 0,C 180,E1 -1078.137,E2 -1078.137} C_VEL
LIN {X 0,Y 594.629,Z 778.589,A -85,B 0,C 180,E1 -1078.645,E2 -1078.645} C_VEL
LIN {X 0,Y 594.678,Z 766.222,A -85,B 0,C 180,E1 -1078.963,E2 -1078.963} C_VEL
LIN {X 0,Y 594.706,Z 752.556,A -85,B 0,C 180,E1 -1079.175,E2 -1079.175} C_VEL
LIN {X 0,Y 594.688,Z 679.801,A -85,B 0,C 180,E1 -1080.063,E2 -1080.063} C_VEL
LIN {X 0,Y 594.428,Z 678.661,A -85,B 0,C 180,E1 -1080.169,E2 -1080.169} C_VEL
LIN {X 0,Y 594.377,Z 678.443,A -85,B 0,C 180,E1 -1081.355,E2 -1081.355} C_VEL
LIN {X 0,Y 594.359,Z 678.453,A -85,B 0,C 180,E1 -1084.068,E2 -1084.068} C_VEL
LIN {X 0,Y 594.385,Z 678.44,A -85,B 0,C 180,E1 -1086.79,E2 -1086.79} C_VEL
LIN {X 0,Y 594.37,Z 678.443,A -85,B 0,C 180,E1 -1089.529,E2 -1089.529} C_VEL
LIN {X 0,Y 594.388,Z 678.45,A -85,B 0,C 180,E1 -1092.288,E2 -1092.288} C_VEL
LIN {X 0,Y 594.371,Z 678.442,A -85,B 0,C 180,E1 -1095.078,E2 -1095.078} C_VEL
LIN {X 0,Y 594.379,Z 678.44,A -85,B 0,C 180,E1 -1097.194,E2 -1097.194} C_VEL
LIN {X 0,Y 594.375,Z 678.444,A -85,B 0,C 180,E1 -1100.054,E2 -1100.054} C_VEL
LIN {X 0,Y 594.361,Z 678.447,A -85,B 0,C 180,E1 -1102.967,E2 -1102.967} C_VEL
LIN {X 0,Y 594.365,Z 678.444,A -85,B 0,C 180,E1 -1105.194,E2 -1105.194} C_VEL
LIN {X 0,Y 594.349,Z 678.444,A -85,B 0,C 180,E1 -1107.518,E2 -1107.518} C_VEL
LIN {X 0,Y 594.392,Z 678.441,A -85,B 0,C 180,E1 -1110.328,E2 -1110.328} C_VEL
LIN {X 0,Y 594.381,Z 678.451,A -85,B 0,C 180,E1 -1112.95,E2 -1112.95} C_VEL
LIN {X 0,Y 594.353,Z 678.447,A -85,B 0,C 180,E1 -1115.409,E2 -1115.409} C_VEL
LIN {X 0,Y 594.386,Z 678.439,A -85,B 0,C 180,E1 -1117.941,E2 -1117.941} C_VEL
LIN {X 0,Y 594.376,Z 678.445,A -85,B 0,C 180,E1 -1120.821,E2 -1120.821} C_VEL
LIN {X 0,Y 594.373,Z 678.452,A -85,B 0,C 180,E1 -1123.299,E2 -1123.299} C_VEL
LIN {X 0,Y 594.365,Z 678.442,A -85,B 0,C 180,E1 -1126.161,E2 -1126.161} C_VEL
LIN {X 0,Y 594.382,Z 678.44,A -85,B 0,C 180,E1 -1128.535,E2 -1128.535} C_VEL
LIN {X 0,Y 594.374,Z 678.447,A -85,B 0,C 180,E1 -1131.297,E2 -1131.297} C_VEL
LIN {X 0,Y 594.353,Z 678.452,A -85,B 0,C 180,E1 -1133.755,E2 -1133.755} C_VEL
LIN {X 0,Y 594.369,Z 678.444,A -85,B 0,C 180,E1 -1136.237,E2 -1136.237} C_VEL
LIN {X 0,Y 594.372,Z 678.442,A -85,B 0,C 180,E1 -1138.649,E2 -1138.649} C_VEL
LIN {X 0,Y 594.384,Z 678.441,A -85,B 0,C 180,E1 -1141.043,E2 -1141.043} C_VEL
LIN {X 0,Y 594.405,Z 678.653,A -85,B 0,C 180,E1 -1143.387,E2 -1143.387} C_VEL
LIN {X 0,Y 595.187,Z 682.049,A -85,B 0,C 180,E1 -1143.82,E2 -1143.82} C_VEL
LIN {X 0,Y 595.023,Z 704.655,A -85,B 0,C 180,E1 -1146.322,E2 -1146.322} C_VEL
LIN {X 0,Y 594.858,Z 733.232,A -85,B 0,C 180,E1 -1149.421,E2 -1149.421} C_VEL
LIN {X 0,Y 594.689,Z 758.447,A -85,B 0,C 180,E1 -1152.105,E2 -1152.105} C_VEL
LIN {X 0,Y 594.551,Z 783.662,A -85,B 0,C 180,E1 -1154.75,E2 -1154.75} C_VEL
LIN {X 0,Y 594.525,Z 802.106,A -85,B 0,C 180,E1 -1156.639,E2 -1156.639} C_VEL
LIN {X 0,Y 594.8,Z 809.431,A -85,B 0,C 180,E1 -1156.743,E2 -1156.743} C_VEL
LIN {X 0,Y 594.653,Z 911.896,A -85,B 0,C 180,E1 -1157.998,E2 -1157.998} C_VEL
LIN {X 0,Y 594.65,Z 925.184,A -85,B 0,C 180,E1 -1158.3,E2 -1158.3} C_VEL
LIN {X 0,Y 594.597,Z 937.551,A -85,B 0,C 180,E1 -1158.718,E2 -1158.718} C_VEL
LIN {X 0,Y 594.538,Z 949.616,A -85,B 0,C 180,E1 -1159.269,E2 -1159.269} C_VEL
LIN {X 0,Y 594.465,Z 961.185,A -85,B 0,C 180,E1 -1159.956,E2 -1159.956} C_VEL
LIN {X 0,Y 594.414,Z 971.584,A -85,B 0,C 180,E1 -1160.729,E2 -1160.729} C_VEL
LIN {X 0,Y 594.348,Z 980.009,A -85,B 0,C 180,E1 -1161.499,E2 -1161.499} C_VEL
LIN {X 0,Y 594.347,Z 987.952,A -85,B 0,C 180,E1 -1162.354,E2 -1162.354} C_VEL
LIN {X 0,Y 594.281,Z 995.819,A -85,B 0,C 180,E1 -1163.409,E2 -1163.409} C_VEL
LIN {X 0,Y 594.289,Z 1002.675,A -85,B 0,C 180,E1 -1164.57,E2 -1164.57} C_VEL
LIN {X 0,Y 594.27,Z 1007.367,A -85,B 0,C 180,E1 -1165.59,E2 -1165.59} C_VEL
LIN {X 0,Y 594.267,Z 1010.953,A -85,B 0,C 180,E1 -1166.609,E2 -1166.609} C_VEL
LIN {X 0,Y 594.226,Z 1012.806,A -85,B 0,C 180,E1 -1167.287,E2 -1167.287} C_VEL
LIN {X 0,Y 594.24,Z 1014.2,A -85,B 0,C 180,E1 -1167.966,E2 -1167.966} C_VEL
LIN {X 0,Y 594.239,Z 1015.783,A -85,B 0,C 180,E1 -1169.321,E2 -1169.321} C_VEL
LIN {X 0,Y 594.236,Z 1016,A -85,B 0,C 180,E1 -1169.999,E2 -1169.999} C_VEL
LIN {X 0,Y 594.247,Z 1015.186,A -85,B 0,C 180,E1 -1171.354,E2 -1171.354} C_VEL
LIN {X 0,Y 594.24,Z 1014.204,A -85,B 0,C 180,E1 -1172.032,E2 -1172.032} C_VEL
LIN {X 0,Y 594.226,Z 1012.812,A -85,B 0,C 180,E1 -1172.711,E2 -1172.711} C_VEL
LIN {X 0,Y 594.288,Z 1009.899,A -85,B 0,C 180,E1 -1173.728,E2 -1173.728} C_VEL
LIN {X 0,Y 594.241,Z 1005.954,A -85,B 0,C 180,E1 -1174.748,E2 -1174.748} C_VEL
LIN {X 0,Y 594.304,Z 999.883,A -85,B 0,C 180,E1 -1175.938,E2 -1175.938} C_VEL
LIN {X 0,Y 594.307,Z 993.243,A -85,B 0,C 180,E1 -1176.961,E2 -1176.961} C_VEL
LIN {X 0,Y 594.359,Z 984.999,A -85,B 0,C 180,E1 -1177.985,E2 -1177.985} C_VEL
LIN {X 0,Y 594.404,Z 974.612,A -85,B 0,C 180,E1 -1179.012,E2 -1179.012} C_VEL
LIN {X 0,Y 594.448,Z 963.763,A -85,B 0,C 180,E1 -1179.87,E2 -1179.87} C_VEL
LIN {X 0,Y 594.507,Z 952.796,A -85,B 0,C 180,E1 -1180.557,E2 -1180.557} C_VEL
LIN {X 0,Y 594.601,Z 940.154,A -85,B 0,C 180,E1 -1181.175,E2 -1181.175} C_VEL
LIN {X 0,Y 594.625,Z 927.533,A -85,B 0,C 180,E1 -1181.633,E2 -1181.633} C_VEL
LIN {X 0,Y 594.667,Z 914.287,A -85,B 0,C 180,E1 -1181.957,E2 -1181.957} C_VEL
LIN {X 0,Y 594.665,Z 893.67,A -85,B 0,C 180,E1 -1182.238,E2 -1182.238} C_VEL
LIN {X 0,Y 594.681,Z 803.342,A -85,B 0,C 180,E1 -1183.333,E2 -1183.333} C_VEL
LIN {X 0,Y 594.513,Z 801.919,A -85,B 0,C 180,E1 -1183.37,E2 -1183.37} C_VEL
LIN {X 0,Y 594.584,Z 775.277,A -85,B 0,C 180,E1 -1186.126,E2 -1186.126} C_VEL
LIN {X 0,Y 594.776,Z 747.654,A -85,B 0,C 180,E1 -1189.038,E2 -1189.038} C_VEL
LIN {X 0,Y 594.892,Z 721.485,A -85,B 0,C 180,E1 -1191.846,E2 -1191.846} C_VEL
LIN {X 0,Y 595.101,Z 696.414,A -85,B 0,C 180,E1 -1194.584,E2 -1194.584} C_VEL
LIN {X 0,Y 595.227,Z 681.963,A -85,B 0,C 180,E1 -1196.187,E2 -1196.187} C_VEL
LIN {X 0,Y 594.4,Z 678.559,A -85,B 0,C 180,E1 -1196.638,E2 -1196.638} C_VEL
LIN {X 0,Y 594.377,Z 678.442,A -85,B 0,C 180,E1 -1198.997,E2 -1198.997} C_VEL
LIN {X 0,Y 594.373,Z 678.443,A -85,B 0,C 180,E1 -1201.642,E2 -1201.642} C_VEL
LIN {X 0,Y 594.374,Z 678.448,A -85,B 0,C 180,E1 -1204.579,E2 -1204.579} C_VEL
LIN {X 0,Y 594.383,Z 678.44,A -85,B 0,C 180,E1 -1207.607,E2 -1207.607} C_VEL
LIN {X 0,Y 594.363,Z 678.453,A -85,B 0,C 180,E1 -1210.566,E2 -1210.566} C_VEL
LIN {X 0,Y 594.36,Z 678.444,A -85,B 0,C 180,E1 -1213.298,E2 -1213.298} C_VEL
LIN {X 0,Y 594.374,Z 678.441,A -85,B 0,C 180,E1 -1216.158,E2 -1216.158} C_VEL
LIN {X 0,Y 594.372,Z 678.446,A -85,B 0,C 180,E1 -1218.535,E2 -1218.535} C_VEL
LIN {X 0,Y 594.382,Z 678.445,A -85,B 0,C 180,E1 -1221.294,E2 -1221.294} C_VEL
LIN {X 0,Y 594.388,Z 678.439,A -85,B 0,C 180,E1 -1223.758,E2 -1223.758} C_VEL
LIN {X 0,Y 594.367,Z 678.441,A -85,B 0,C 180,E1 -1226.238,E2 -1226.238} C_VEL
LIN {X 0,Y 594.359,Z 678.444,A -85,B 0,C 180,E1 -1228.649,E2 -1228.649} C_VEL
LIN {X 0,Y 594.376,Z 678.446,A -85,B 0,C 180,E1 -1231.041,E2 -1231.041} C_VEL
LIN {X 0,Y 594.381,Z 678.442,A -85,B 0,C 180,E1 -1233.975,E2 -1233.975} C_VEL
LIN {X 0,Y 594.383,Z 678.44,A -85,B 0,C 180,E1 -1236.296,E2 -1236.296} C_VEL
LIN {X 0,Y 594.393,Z 678.442,A -85,B 0,C 180,E1 -1239.224,E2 -1239.224} C_VEL
LIN {X 0,Y 594.369,Z 678.445,A -85,B 0,C 180,E1 -1242.095,E2 -1242.095} C_VEL
LIN {X 0,Y 594.36,Z 678.446,A -85,B 0,C 180,E1 -1244.219,E2 -1244.219} C_VEL
LIN {X 0,Y 594.351,Z 678.443,A -85,B 0,C 180,E1 -1247.017,E2 -1247.017} C_VEL
LIN {X 0,Y 594.383,Z 678.447,A -85,B 0,C 180,E1 -1249.784,E2 -1249.784} C_VEL
LIN {X 0,Y 594.41,Z 678.439,A -85,B 0,C 180,E1 -1252.527,E2 -1252.527} C_VEL
LIN {X 0,Y 594.372,Z 678.44,A -85,B 0,C 180,E1 -1255.252,E2 -1255.252} C_VEL
LIN {X 0,Y 594.378,Z 678.445,A -85,B 0,C 180,E1 -1257.967,E2 -1257.967} C_VEL
LIN {X 0,Y 594.42,Z 678.44,A -85,B 0,C 180,E1 -1260.678,E2 -1260.678} C_VEL
LIN {X 0,Y 594.372,Z 678.44,A -85,B 0,C 180,E1 -1263.39,E2 -1263.39} C_VEL
LIN {X 0,Y 594.384,Z 678.439,A -85,B 0,C 180,E1 -1265.428,E2 -1265.428} C_VEL
LIN {X 0,Y 594.399,Z 678.44,A -85,B 0,C 180,E1 -1268.157,E2 -1268.157} C_VEL
LIN {X 0,Y 594.384,Z 678.444,A -85,B 0,C 180,E1 -1271.078,E2 -1271.078} C_VEL
LIN {X 0,Y 594.366,Z 678.441,A -85,B 0,C 180,E1 -1273.68,E2 -1273.68} C_VEL
LIN {X 0,Y 594.349,Z 678.447,A -85,B 0,C 180,E1 -1275.338,E2 -1275.338} C_VEL
LIN {X 0,Y 593.673,Z 678.53,A -85,B 0,C 180,E1 -1275.904,E2 -1275.904} C_VEL
LIN {X 0,Y 590.802,Z 678.894,A -85,B 0,C 180,E1 -1276.822,E2 -1276.822} C_VEL
LIN {X 0,Y 588.389,Z 679.189,A -85,B 0,C 180,E1 -1277.561,E2 -1277.561} C_VEL
LIN {X 0,Y 587.367,Z 679.313,A -85,B 0,C 180,E1 -1278.131,E2 -1278.131} C_VEL
LIN {X 0,Y 587.292,Z 679.324,A -85,B 0,C 180,E1 -1278.324,E2 -1278.324} C_VEL
LIN {X 0,Y 587.319,Z 679.329,A -85,B 0,C 180,E1 -1281.038,E2 -1281.038} C_VEL
LIN {X 0,Y 587.309,Z 679.33,A -85,B 0,C 180,E1 -1283.26,E2 -1283.26} C_VEL
LIN {X 0,Y 587.328,Z 679.325,A -85,B 0,C 180,E1 -1285.517,E2 -1285.517} C_VEL
LIN {X 0,Y 587.334,Z 679.32,A -85,B 0,C 180,E1 -1287.819,E2 -1287.819} C_VEL
LIN {X 0,Y 587.325,Z 679.319,A -85,B 0,C 180,E1 -1290.511,E2 -1290.511} C_VEL
LIN {X 0,Y 587.329,Z 679.326,A -85,B 0,C 180,E1 -1293.397,E2 -1293.397} C_VEL
LIN {X 0,Y 587.297,Z 679.328,A -85,B 0,C 180,E1 -1295.9,E2 -1295.9} C_VEL
LIN {X 0,Y 587.32,Z 679.319,A -85,B 0,C 180,E1 -1298.481,E2 -1298.481} C_VEL
LIN {X 0,Y 587.324,Z 679.32,A -85,B 0,C 180,E1 -1301.158,E2 -1301.158} C_VEL
LIN {X 0,Y 587.32,Z 679.328,A -85,B 0,C 180,E1 -1304.115,E2 -1304.115} C_VEL
LIN {X 0,Y 587.289,Z 679.323,A -85,B 0,C 180,E1 -1306.993,E2 -1306.993} C_VEL
LIN {X 0,Y 587.302,Z 679.327,A -85,B 0,C 180,E1 -1309.746,E2 -1309.746} C_VEL
LIN {X 0,Y 587.345,Z 679.48,A -85,B 0,C 180,E1 -1311.761,E2 -1311.761} C_VEL
LIN {X 0,Y 587.664,Z 680.727,A -85,B 0,C 180,E1 -1311.882,E2 -1311.882} C_VEL
LIN {X 0,Y 587.837,Z 697.792,A -85,B 0,C 180,E1 -1312.1,E2 -1312.1} C_VEL
LIN {X 0,Y 587.757,Z 762.432,A -85,B 0,C 180,E1 -1312.91,E2 -1312.91} C_VEL
LIN {X 0,Y 587.705,Z 775.729,A -85,B 0,C 180,E1 -1313.221,E2 -1313.221} C_VEL
LIN {X 0,Y 587.596,Z 788.05,A -85,B 0,C 180,E1 -1313.646,E2 -1313.646} C_VEL
LIN {X 0,Y 587.537,Z 800.141,A -85,B 0,C 180,E1 -1314.214,E2 -1314.214} C_VEL
LIN {X 0,Y 587.429,Z 812.262,A -85,B 0,C 180,E1 -1314.953,E2 -1314.953} C_VEL
LIN {X 0,Y 587.363,Z 823.015,A -85,B 0,C 180,E1 -1315.782,E2 -1315.782} C_VEL
LIN {X 0,Y 587.305,Z 831.624,A -85,B 0,C 180,E1 -1316.603,E2 -1316.603} C_VEL
LIN {X 0,Y 587.277,Z 840.442,A -85,B 0,C 180,E1 -1317.622,E2 -1317.622} C_VEL
LIN {X 0,Y 587.238,Z 847.465,A -85,B 0,C 180,E1 -1318.629,E2 -1318.629} C_VEL
LIN {X 0,Y 587.185,Z 854.029,A -85,B 0,C 180,E1 -1319.823,E2 -1319.823} C_VEL
LIN {X 0,Y 587.17,Z 858.578,A -85,B 0,C 180,E1 -1320.899,E2 -1320.899} C_VEL
LIN {X 0,Y 587.157,Z 862.486,A -85,B 0,C 180,E1 -1322.174,E2 -1322.174} C_VEL
LIN {X 0,Y 587.13,Z 864.132,A -85,B 0,C 180,E1 -1322.945,E2 -1322.945} C_VEL
LIN {X 0,Y 587.119,Z 865.407,A -85,B 0,C 180,E1 -1323.868,E2 -1323.868} C_VEL
LIN {X 0,Y 587.117,Z 865.862,A -85,B 0,C 180,E1 -1324.475,E2 -1324.475} C_VEL
LIN {X 0,Y 587.135,Z 865.91,A -85,B 0,C 180,E1 -1325.468,E2 -1325.468} C_VEL
LIN {X 0,Y 587.115,Z 864.793,A -85,B 0,C 180,E1 -1326.734,E2 -1326.734} C_VEL
LIN {X 0,Y 587.146,Z 863.47,A -85,B 0,C 180,E1 -1327.48,E2 -1327.48} C_VEL
LIN {X 0,Y 587.157,Z 860.609,A -85,B 0,C 180,E1 -1328.589,E2 -1328.589} C_VEL
LIN {X 0,Y 587.203,Z 856.608,A -85,B 0,C 180,E1 -1329.692,E2 -1329.692} C_VEL
LIN {X 0,Y 587.228,Z 851.573,A -85,B 0,C 180,E1 -1330.75,E2 -1330.75} C_VEL
LIN {X 0,Y 587.223,Z 844.8,A -85,B 0,C 180,E1 -1331.871,E2 -1331.871} C_VEL
LIN {X 0,Y 587.269,Z 836.565,A -85,B 0,C 180,E1 -1332.945,E2 -1332.945} C_VEL
LIN {X 0,Y 587.355,Z 826.171,A -85,B 0,C 180,E1 -1334.027,E2 -1334.027} C_VEL
LIN {X 0,Y 587.416,Z 815.338,A -85,B 0,C 180,E1 -1334.918,E2 -1334.918} C_VEL
LIN {X 0,Y 587.501,Z 805.59,A -85,B 0,C 180,E1 -1335.566,E2 -1335.566} C_VEL
LIN {X 0,Y 587.573,Z 794.509,A -85,B 0,C 180,E1 -1336.161,E2 -1336.161} C_VEL
LIN {X 0,Y 587.644,Z 782.701,A -85,B 0,C 180,E1 -1336.647,E2 -1336.647} C_VEL
LIN {X 0,Y 587.707,Z 769.978,A -85,B 0,C 180,E1 -1337.022,E2 -1337.022} C_VEL
LIN {X 0,Y 587.76,Z 756.909,A -85,B 0,C 180,E1 -1337.265,E2 -1337.265} C_VEL
LIN {X 0,Y 587.776,Z 681.221,A -85,B 0,C 180,E1 -1338.196,E2 -1338.196} C_VEL
LIN {X 0,Y 587.419,Z 679.857,A -85,B 0,C 180,E1 -1338.266,E2 -1338.266} C_VEL
LIN {X 0,Y 587.333,Z 679.334,A -85,B 0,C 180,E1 -1338.439,E2 -1338.439} C_VEL
LIN {X 0,Y 587.302,Z 679.323,A -85,B 0,C 180,E1 -1341.052,E2 -1341.052} C_VEL
LIN {X 0,Y 587.313,Z 679.327,A -85,B 0,C 180,E1 -1343.818,E2 -1343.818} C_VEL
LIN {X 0,Y 587.307,Z 679.328,A -85,B 0,C 180,E1 -1345.884,E2 -1345.884} C_VEL
LIN {X 0,Y 587.303,Z 679.325,A -85,B 0,C 180,E1 -1348.63,E2 -1348.63} C_VEL
LIN {X 0,Y 587.288,Z 679.327,A -85,B 0,C 180,E1 -1350.687,E2 -1350.687} C_VEL
LIN {X 0,Y 587.346,Z 679.32,A -85,B 0,C 180,E1 -1352.744,E2 -1352.744} C_VEL
LIN {X 0,Y 587.317,Z 679.32,A -85,B 0,C 180,E1 -1355.494,E2 -1355.494} C_VEL
LIN {X 0,Y 587.318,Z 679.326,A -85,B 0,C 180,E1 -1358.257,E2 -1358.257} C_VEL
LIN {X 0,Y 587.303,Z 679.324,A -85,B 0,C 180,E1 -1361.108,E2 -1361.108} C_VEL
LIN {X 0,Y 587.326,Z 679.318,A -85,B 0,C 180,E1 -1363.847,E2 -1363.847} C_VEL
LIN {X 0,Y 587.314,Z 679.331,A -85,B 0,C 180,E1 -1366.801,E2 -1366.801} C_VEL
LIN {X 0,Y 587.296,Z 679.322,A -85,B 0,C 180,E1 -1369.578,E2 -1369.578} C_VEL
LIN {X 0,Y 587.3,Z 679.322,A -85,B 0,C 180,E1 -1371.776,E2 -1371.776} C_VEL
LIN {X 0,Y 587.289,Z 679.327,A -85,B 0,C 180,E1 -1374.565,E2 -1374.565} C_VEL
LIN {X 0,Y 587.302,Z 679.331,A -85,B 0,C 180,E1 -1377.048,E2 -1377.048} C_VEL
LIN {X 0,Y 587.288,Z 679.33,A -85,B 0,C 180,E1 -1379.384,E2 -1379.384} C_VEL
LIN {X 0,Y 587.3,Z 679.323,A -85,B 0,C 180,E1 -1381.828,E2 -1381.828} C_VEL
LIN {X 0,Y 587.288,Z 679.321,A -85,B 0,C 180,E1 -1384.338,E2 -1384.338} C_VEL
LIN {X 0,Y 587.31,Z 679.327,A -85,B 0,C 180,E1 -1387.611,E2 -1387.611} C_VEL
LIN {X 0,Y 587.279,Z 679.325,A -85,B 0,C 180,E1 -1390.258,E2 -1390.258} C_VEL
LIN {X 0,Y 587.278,Z 679.328,A -85,B 0,C 180,E1 -1393.114,E2 -1393.114} C_VEL
LIN {X 0,Y 587.276,Z 679.329,A -85,B 0,C 180,E1 -1396.045,E2 -1396.045} C_VEL
LIN {X 0,Y 587.275,Z 679.325,A -85,B 0,C 180,E1 -1398.933,E2 -1398.933} C_VEL
LIN {X 0,Y 587.276,Z 679.33,A -85,B 0,C 180,E1 -1401.516,E2 -1401.516} C_VEL
LIN {X 0,Y 587.256,Z 679.33,A -85,B 0,C 180,E1 -1404.469,E2 -1404.469} C_VEL
LIN {X 0,Y 587.283,Z 679.324,A -85,B 0,C 180,E1 -1406.898,E2 -1406.898} C_VEL
LIN {X 0,Y 587.314,Z 679.327,A -85,B 0,C 180,E1 -1409.828,E2 -1409.828} C_VEL
LIN {X 0,Y 587.293,Z 679.324,A -85,B 0,C 180,E1 -1412.952,E2 -1412.952} C_VEL
LIN {X 0,Y 587.37,Z 679.563,A -85,B 0,C 180,E1 -1413.781,E2 -1413.781} C_VEL
LIN {X 0,Y 587.608,Z 680.618,A -85,B 0,C 180,E1 -1413.878,E2 -1413.878} C_VEL
LIN {X 0,Y 587.832,Z 688.316,A -85,B 0,C 180,E1 -1413.983,E2 -1413.983} C_VEL
LIN {X 0,Y 587.71,Z 762.051,A -85,B 0,C 180,E1 -1414.903,E2 -1414.903} C_VEL
LIN {X 0,Y 587.685,Z 774.861,A -85,B 0,C 180,E1 -1415.197,E2 -1415.197} C_VEL
LIN {X 0,Y 587.586,Z 787.08,A -85,B 0,C 180,E1 -1415.611,E2 -1415.611} C_VEL
LIN {X 0,Y 587.532,Z 799.695,A -85,B 0,C 180,E1 -1416.189,E2 -1416.189} C_VEL
LIN {X 0,Y 587.451,Z 811.04,A -85,B 0,C 180,E1 -1416.87,E2 -1416.87} C_VEL
LIN {X 0,Y 587.397,Z 821.734,A -85,B 0,C 180,E1 -1417.674,E2 -1417.674} C_VEL
LIN {X 0,Y 587.311,Z 829.693,A -85,B 0,C 180,E1 -1418.409,E2 -1418.409} C_VEL
LIN {X 0,Y 587.286,Z 838.091,A -85,B 0,C 180,E1 -1419.327,E2 -1419.327} C_VEL
LIN {X 0,Y 587.227,Z 844.904,A -85,B 0,C 180,E1 -1420.239,E2 -1420.239} C_VEL
LIN {X 0,Y 587.233,Z 850.518,A -85,B 0,C 180,E1 -1421.147,E2 -1421.147} C_VEL
LIN {X 0,Y 587.171,Z 855.882,A -85,B 0,C 180,E1 -1422.229,E2 -1422.229} C_VEL
LIN {X 0,Y 587.172,Z 859.986,A -85,B 0,C 180,E1 -1423.306,E2 -1423.306} C_VEL
LIN {X 0,Y 587.158,Z 862.089,A -85,B 0,C 180,E1 -1424.02,E2 -1424.02} C_VEL
LIN {X 0,Y 587.132,Z 863.721,A -85,B 0,C 180,E1 -1424.731,E2 -1424.731} C_VEL
LIN {X 0,Y 587.164,Z 865.35,A -85,B 0,C 180,E1 -1425.82,E2 -1425.82} C_VEL
LIN {X 0,Y 587.145,Z 865.963,A -85,B 0,C 180,E1 -1426.854,E2 -1426.854} C_VEL
LIN {X 0,Y 587.16,Z 865.865,A -85,B 0,C 180,E1 -1427.558,E2 -1427.558} C_VEL
LIN {X 0,Y 587.156,Z 865.363,A -85,B 0,C 180,E1 -1428.259,E2 -1428.259} C_VEL
LIN {X 0,Y 587.17,Z 864.432,A -85,B 0,C 180,E1 -1428.959,E2 -1428.959} C_VEL
LIN {X 0,Y 587.141,Z 863.092,A -85,B 0,C 180,E1 -1429.656,E2 -1429.656} C_VEL
LIN {X 0,Y 587.189,Z 860.258,A -85,B 0,C 180,E1 -1430.701,E2 -1430.701} C_VEL
LIN {X 0,Y 587.19,Z 856.394,A -85,B 0,C 180,E1 -1431.742,E2 -1431.742} C_VEL
LIN {X 0,Y 587.216,Z 851.397,A -85,B 0,C 180,E1 -1432.781,E2 -1432.781} C_VEL
LIN {X 0,Y 587.218,Z 845.137,A -85,B 0,C 180,E1 -1433.816,E2 -1433.816} C_VEL
LIN {X 0,Y 587.305,Z 837.378,A -85,B 0,C 180,E1 -1434.851,E2 -1434.851} C_VEL
LIN {X 0,Y 587.322,Z 827.71,A -85,B 0,C 180,E1 -1435.883,E2 -1435.883} C_VEL
LIN {X 0,Y 587.39,Z 817.67,A -85,B 0,C 180,E1 -1436.742,E2 -1436.742} C_VEL
LIN {X 0,Y 587.477,Z 807.799,A -85,B 0,C 180,E1 -1437.429,E2 -1437.429} C_VEL
LIN {X 0,Y 587.526,Z 797.13,A -85,B 0,C 180,E1 -1438.029,E2 -1438.029} C_VEL
LIN {X 0,Y 587.632,Z 785.414,A -85,B 0,C 180,E1 -1438.544,E2 -1438.544} C_VEL
LIN {X 0,Y 587.697,Z 772.845,A -85,B 0,C 180,E1 -1438.951,E2 -1438.951} C_VEL
LIN {X 0,Y 587.733,Z 759.474,A -85,B 0,C 180,E1 -1439.229,E2 -1439.229} C_VEL
LIN {X 0,Y 587.718,Z 680.87,A -85,B 0,C 180,E1 -1440.206,E2 -1440.206} C_VEL
LIN {X 0,Y 587.418,Z 679.625,A -85,B 0,C 180,E1 -1440.3,E2 -1440.3} C_VEL
LIN {X 0,Y 587.385,Z 679.313,A -85,B 0,C 180,E1 -1440.685,E2 -1440.685} C_VEL
LIN {X 0,Y 587.336,Z 679.321,A -85,B 0,C 180,E1 -1443.43,E2 -1443.43} C_VEL
LIN {X 0,Y 587.314,Z 679.33,A -85,B 0,C 180,E1 -1446.182,E2 -1446.182} C_VEL
LIN {X 0,Y 587.345,Z 679.326,A -85,B 0,C 180,E1 -1448.255,E2 -1448.255} C_VEL
LIN {X 0,Y 587.356,Z 679.315,A -85,B 0,C 180,E1 -1451.133,E2 -1451.133} C_VEL
LIN {X 0,Y 587.371,Z 679.323,A -85,B 0,C 180,E1 -1454.26,E2 -1454.26} C_VEL
LIN {X 0,Y 587.317,Z 679.32,A -85,B 0,C 180,E1 -1457.407,E2 -1457.407} C_VEL
LIN {X 0,Y 587.316,Z 679.32,A -85,B 0,C 180,E1 -1459.576,E2 -1459.576} C_VEL
LIN {X 0,Y 587.32,Z 679.32,A -85,B 0,C 180,E1 -1461.774,E2 -1461.774} C_VEL
LIN {X 0,Y 587.353,Z 679.325,A -85,B 0,C 180,E1 -1464.758,E2 -1464.758} C_VEL
LIN {X 0,Y 587.317,Z 679.325,A -85,B 0,C 180,E1 -1467.047,E2 -1467.047} C_VEL
LIN {X 0,Y 587.351,Z 679.318,A -85,B 0,C 180,E1 -1469.379,E2 -1469.379} C_VEL
LIN {X 0,Y 587.346,Z 679.316,A -85,B 0,C 180,E1 -1471.834,E2 -1471.834} C_VEL
LIN {X 0,Y 587.347,Z 679.317,A -85,B 0,C 180,E1 -1474.346,E2 -1474.346} C_VEL
LIN {X 0,Y 587.348,Z 679.318,A -85,B 0,C 180,E1 -1477.608,E2 -1477.608} C_VEL
LIN {X 0,Y 587.314,Z 679.32,A -85,B 0,C 180,E1 -1480.255,E2 -1480.255} C_VEL
LIN {X 0,Y 587.322,Z 679.328,A -85,B 0,C 180,E1 -1483.118,E2 -1483.118} C_VEL
LIN {X 0,Y 587.318,Z 679.321,A -85,B 0,C 180,E1 -1486.048,E2 -1486.048} C_VEL
LIN {X 0,Y 587.34,Z 679.32,A -85,B 0,C 180,E1 -1488.925,E2 -1488.925} C_VEL
LIN {X 0,Y 587.323,Z 679.33,A -85,B 0,C 180,E1 -1491.519,E2 -1491.519} C_VEL
LIN {X 0,Y 587.294,Z 679.326,A -85,B 0,C 180,E1 -1494.099,E2 -1494.099} C_VEL
LIN {X 0,Y 587.342,Z 679.317,A -85,B 0,C 180,E1 -1496.888,E2 -1496.888} C_VEL
LIN {X 0,Y 587.336,Z 679.328,A -85,B 0,C 180,E1 -1499.829,E2 -1499.829} C_VEL
LIN {X 0,Y 587.309,Z 679.328,A -85,B 0,C 180,E1 -1502.316,E2 -1502.316} C_VEL
LIN {X 0,Y 587.388,Z 679.546,A -85,B 0,C 180,E1 -1503.148,E2 -1503.148} C_VEL
LIN {X 0,Y 588.448,Z 684.483,A -85,B 0,C 180,E1 -1503.774,E2 -1503.774} C_VEL
LIN {X 0,Y 588.212,Z 706.336,A -85,B 0,C 180,E1 -1506.218,E2 -1506.218} C_VEL
LIN {X 0,Y 587.965,Z 734.913,A -85,B 0,C 180,E1 -1509.352,E2 -1509.352} C_VEL
LIN {X 0,Y 587.749,Z 760.128,A -85,B 0,C 180,E1 -1512.066,E2 -1512.066} C_VEL
LIN {X 0,Y 587.558,Z 787.024,A -85,B 0,C 180,E1 -1514.92,E2 -1514.92} C_VEL
LIN {X 0,Y 587.517,Z 801.883,A -85,B 0,C 180,E1 -1516.466,E2 -1516.466} C_VEL
LIN {X 0,Y 587.86,Z 805.854,A -85,B 0,C 180,E1 -1516.54,E2 -1516.54} C_VEL
LIN {X 0,Y 587.716,Z 911.896,A -85,B 0,C 180,E1 -1517.854,E2 -1517.854} C_VEL
LIN {X 0,Y 587.7,Z 925.185,A -85,B 0,C 180,E1 -1518.16,E2 -1518.16} C_VEL
LIN {X 0,Y 587.629,Z 937.733,A -85,B 0,C 180,E1 -1518.589,E2 -1518.589} C_VEL
LIN {X 0,Y 587.561,Z 949.615,A -85,B 0,C 180,E1 -1519.14,E2 -1519.14} C_VEL
LIN {X 0,Y 587.462,Z 961.186,A -85,B 0,C 180,E1 -1519.835,E2 -1519.835} C_VEL
LIN {X 0,Y 587.392,Z 971.585,A -85,B 0,C 180,E1 -1520.617,E2 -1520.617} C_VEL
LIN {X 0,Y 587.299,Z 980.018,A -85,B 0,C 180,E1 -1521.396,E2 -1521.396} C_VEL
LIN {X 0,Y 587.274,Z 987.952,A -85,B 0,C 180,E1 -1522.262,E2 -1522.262} C_VEL
LIN {X 0,Y 587.231,Z 994.463,A -85,B 0,C 180,E1 -1523.125,E2 -1523.125} C_VEL
LIN {X 0,Y 587.236,Z 1000.861,A -85,B 0,C 180,E1 -1524.16,E2 -1524.16} C_VEL
LIN {X 0,Y 587.147,Z 1005.946,A -85,B 0,C 180,E1 -1525.193,E2 -1525.193} C_VEL
LIN {X 0,Y 587.212,Z 1009.893,A -85,B 0,C 180,E1 -1526.225,E2 -1526.225} C_VEL
LIN {X 0,Y 587.132,Z 1012.806,A -85,B 0,C 180,E1 -1527.255,E2 -1527.255} C_VEL
LIN {X 0,Y 587.139,Z 1014.199,A -85,B 0,C 180,E1 -1527.941,E2 -1527.941} C_VEL
LIN {X 0,Y 587.14,Z 1015.783,A -85,B 0,C 180,E1 -1529.313,E2 -1529.313} C_VEL
LIN {X 0,Y 587.137,Z 1016,A -85,B 0,C 180,E1 -1529.999,E2 -1529.999} C_VEL
LIN {X 0,Y 587.147,Z 1015.186,A -85,B 0,C 180,E1 -1531.371,E2 -1531.371} C_VEL
LIN {X 0,Y 587.139,Z 1014.203,A -85,B 0,C 180,E1 -1532.057,E2 -1532.057} C_VEL
LIN {X 0,Y 587.132,Z 1012.812,A -85,B 0,C 180,E1 -1532.743,E2 -1532.743} C_VEL
LIN {X 0,Y 587.212,Z 1009.899,A -85,B 0,C 180,E1 -1533.773,E2 -1533.773} C_VEL
LIN {X 0,Y 587.147,Z 1005.954,A -85,B 0,C 180,E1 -1534.805,E2 -1534.805} C_VEL
LIN {X 0,Y 587.217,Z 999.884,A -85,B 0,C 180,E1 -1536.01,E2 -1536.01} C_VEL
LIN {X 0,Y 587.244,Z 993.244,A -85,B 0,C 180,E1 -1537.045,E2 -1537.045} C_VEL
LIN {X 0,Y 587.297,Z 984.999,A -85,B 0,C 180,E1 -1538.082,E2 -1538.082} C_VEL
LIN {X 0,Y 587.356,Z 974.612,A -85,B 0,C 180,E1 -1539.121,E2 -1539.121} C_VEL
LIN {X 0,Y 587.444,Z 963.763,A -85,B 0,C 180,E1 -1539.989,E2 -1539.989} C_VEL
LIN {X 0,Y 587.524,Z 952.797,A -85,B 0,C 180,E1 -1540.684,E2 -1540.684} C_VEL
LIN {X 0,Y 587.617,Z 941.191,A -85,B 0,C 180,E1 -1541.264,E2 -1541.264} C_VEL
LIN {X 0,Y 587.658,Z 928.909,A -85,B 0,C 180,E1 -1541.729,E2 -1541.729} C_VEL
LIN {X 0,Y 587.698,Z 916.567,A -85,B 0,C 180,E1 -1542.057,E2 -1542.057} C_VEL
LIN {X 0,Y 587.756,Z 900.825,A -85,B 0,C 180,E1 -1542.296,E2 -1542.296} C_VEL
LIN {X 0,Y 587.723,Z 803.565,A -85,B 0,C 180,E1 -1543.492,E2 -1543.492} C_VEL
LIN {X 0,Y 587.496,Z 801.66,A -85,B 0,C 180,E1 -1543.555,E2 -1543.555} C_VEL
LIN {X 0,Y 587.649,Z 775.277,A -85,B 0,C 180,E1 -1546.322,E2 -1546.322} C_VEL
LIN {X 0,Y 587.869,Z 747.346,A -85,B 0,C 180,E1 -1549.304,E2 -1549.304} C_VEL
LIN {X 0,Y 588.033,Z 723.166,A -85,B 0,C 180,E1 -1551.93,E2 -1551.93} C_VEL
LIN {X 0,Y 588.202,Z 702.994,A -85,B 0,C 180,E1 -1554.155,E2 -1554.155} C_VEL
LIN {X 0,Y 588.471,Z 684.503,A -85,B 0,C 180,E1 -1556.223,E2 -1556.223} C_VEL
LIN {X 0,Y 587.347,Z 679.463,A -85,B 0,C 180,E1 -1556.876,E2 -1556.876} C_VEL
LIN {X 0,Y 587.342,Z 679.319,A -85,B 0,C 180,E1 -1559.378,E2 -1559.378} C_VEL
LIN {X 0,Y 587.341,Z 679.321,A -85,B 0,C 180,E1 -1561.835,E2 -1561.835} C_VEL
LIN {X 0,Y 587.338,Z 679.327,A -85,B 0,C 180,E1 -1564.346,E2 -1564.346} C_VEL
LIN {X 0,Y 587.338,Z 679.317,A -85,B 0,C 180,E1 -1567.607,E2 -1567.607} C_VEL
LIN {X 0,Y 587.306,Z 679.326,A -85,B 0,C 180,E1 -1570.253,E2 -1570.253} C_VEL
LIN {X 0,Y 587.309,Z 679.324,A -85,B 0,C 180,E1 -1573.117,E2 -1573.117} C_VEL
LIN {X 0,Y 587.327,Z 679.319,A -85,B 0,C 180,E1 -1576.05,E2 -1576.05} C_VEL
LIN {X 0,Y 587.329,Z 679.328,A -85,B 0,C 180,E1 -1578.924,E2 -1578.924} C_VEL
LIN {X 0,Y 587.327,Z 679.321,A -85,B 0,C 180,E1 -1581.52,E2 -1581.52} C_VEL
LIN {X 0,Y 587.342,Z 679.317,A -85,B 0,C 180,E1 -1584.454,E2 -1584.454} C_VEL
LIN {X 0,Y 587.329,Z 679.324,A -85,B 0,C 180,E1 -1586.887,E2 -1586.887} C_VEL
LIN {X 0,Y 587.336,Z 679.32,A -85,B 0,C 180,E1 -1589.83,E2 -1589.83} C_VEL
LIN {X 0,Y 587.341,Z 679.316,A -85,B 0,C 180,E1 -1592.306,E2 -1592.306} C_VEL
LIN {X 0,Y 587.326,Z 679.318,A -85,B 0,C 180,E1 -1594.483,E2 -1594.483} C_VEL
LIN {X 0,Y 587.308,Z 679.325,A -85,B 0,C 180,E1 -1597.131,E2 -1597.131} C_VEL
LIN {X 0,Y 587.322,Z 679.329,A -85,B 0,C 180,E1 -1599.695,E2 -1599.695} C_VEL
LIN {X 0,Y 587.34,Z 679.316,A -85,B 0,C 180,E1 -1602.594,E2 -1602.594} C_VEL
LIN {X 0,Y 587.353,Z 679.324,A -85,B 0,C 180,E1 -1605.739,E2 -1605.739} C_VEL
LIN {X 0,Y 587.335,Z 679.317,A -85,B 0,C 180,E1 -1608.866,E2 -1608.866} C_VEL
LIN {X 0,Y 587.355,Z 679.319,A -85,B 0,C 180,E1 -1611.745,E2 -1611.745} C_VEL
LIN {X 0,Y 587.363,Z 679.318,A -85,B 0,C 180,E1 -1614.507,E2 -1614.507} C_VEL
LIN {X 0,Y 587.356,Z 679.314,A -85,B 0,C 180,E1 -1617.257,E2 -1617.257} C_VEL
LIN {X 0,Y 587.364,Z 679.318,A -85,B 0,C 180,E1 -1620,E2 -1620} C_VEL
LIN {X 0,Y 587.374,Z 679.318,A -85,B 0,C 180,E1 -1622.743,E2 -1622.743} C_VEL
LIN {X 0,Y 587.347,Z 679.315,A -85,B 0,C 180,E1 -1625.493,E2 -1625.493} C_VEL
LIN {X 0,Y 587.356,Z 679.319,A -85,B 0,C 180,E1 -1628.256,E2 -1628.256} C_VEL
LIN {X 0,Y 587.351,Z 679.319,A -85,B 0,C 180,E1 -1631.142,E2 -1631.142} C_VEL
LIN {X 0,Y 587.345,Z 679.318,A -85,B 0,C 180,E1 -1634.258,E2 -1634.258} C_VEL
LIN {X 0,Y 587.337,Z 679.321,A -85,B 0,C 180,E1 -1637.407,E2 -1637.407} C_VEL
LIN {X 0,Y 587.292,Z 679.324,A -85,B 0,C 180,E1 -1638.324,E2 -1638.324} C_VEL
LIN {X 0,Y 586.652,Z 679.411,A -85,B 0,C 180,E1 -1638.896,E2 -1638.896} C_VEL
LIN {X 0,Y 583.83,Z 679.768,A -85,B 0,C 180,E1 -1639.825,E2 -1639.825} C_VEL
LIN {X 0,Y 581.419,Z 680.069,A -85,B 0,C 180,E1 -1640.572,E2 -1640.572} C_VEL
LIN {X 0,Y 580.365,Z 680.196,A -85,B 0,C 180,E1 -1641.148,E2 -1641.148} C_VEL
LIN {X 0,Y 580.269,Z 680.204,A -85,B 0,C 180,E1 -1641.343,E2 -1641.343} C_VEL
LIN {X 0,Y 580.262,Z 680.202,A -85,B 0,C 180,E1 -1643.559,E2 -1643.559} C_VEL
LIN {X 0,Y 580.276,Z 680.197,A -85,B 0,C 180,E1 -1646.334,E2 -1646.334} C_VEL
LIN {X 0,Y 580.289,Z 680.203,A -85,B 0,C 180,E1 -1649.31,E2 -1649.31} C_VEL
LIN {X 0,Y 580.287,Z 680.195,A -85,B 0,C 180,E1 -1652.202,E2 -1652.202} C_VEL
LIN {X 0,Y 580.279,Z 680.196,A -85,B 0,C 180,E1 -1654.697,E2 -1654.697} C_VEL
LIN {X 0,Y 580.29,Z 680.199,A -85,B 0,C 180,E1 -1657.269,E2 -1657.269} C_VEL
LIN {X 0,Y 580.283,Z 680.199,A -85,B 0,C 180,E1 -1660.272,E2 -1660.272} C_VEL
LIN {X 0,Y 580.269,Z 680.198,A -85,B 0,C 180,E1 -1662.708,E2 -1662.708} C_VEL
LIN {X 0,Y 580.252,Z 680.205,A -85,B 0,C 180,E1 -1665.611,E2 -1665.611} C_VEL
LIN {X 0,Y 580.268,Z 680.206,A -85,B 0,C 180,E1 -1668.232,E2 -1668.232} C_VEL
LIN {X 0,Y 580.267,Z 680.205,A -85,B 0,C 180,E1 -1670.966,E2 -1670.966} C_VEL
LIN {X 0,Y 580.336,Z 680.37,A -85,B 0,C 180,E1 -1671.612,E2 -1671.612} C_VEL
LIN {X 0,Y 580.586,Z 681.625,A -85,B 0,C 180,E1 -1671.73,E2 -1671.73} C_VEL
LIN {X 0,Y 580.945,Z 683.951,A -85,B 0,C 180,E1 -1671.771,E2 -1671.771} C_VEL
LIN {X 0,Y 580.834,Z 762.258,A -85,B 0,C 180,E1 -1672.76,E2 -1672.76} C_VEL
LIN {X 0,Y 580.738,Z 775.865,A -85,B 0,C 180,E1 -1673.081,E2 -1673.081} C_VEL
LIN {X 0,Y 580.621,Z 788.434,A -85,B 0,C 180,E1 -1673.522,E2 -1673.522} C_VEL
LIN {X 0,Y 580.559,Z 800.648,A -85,B 0,C 180,E1 -1674.11,E2 -1674.11} C_VEL
LIN {X 0,Y 580.453,Z 811.644,A -85,B 0,C 180,E1 -1674.787,E2 -1674.787} C_VEL
LIN {X 0,Y 580.371,Z 821.981,A -85,B 0,C 180,E1 -1675.58,E2 -1675.58} C_VEL
LIN {X 0,Y 580.257,Z 831.139,A -85,B 0,C 180,E1 -1676.448,E2 -1676.448} C_VEL
LIN {X 0,Y 580.228,Z 839.311,A -85,B 0,C 180,E1 -1677.386,E2 -1677.386} C_VEL
LIN {X 0,Y 580.186,Z 845.856,A -85,B 0,C 180,E1 -1678.299,E2 -1678.299} C_VEL
LIN {X 0,Y 580.124,Z 852.333,A -85,B 0,C 180,E1 -1679.417,E2 -1679.417} C_VEL
LIN {X 0,Y 580.109,Z 857.265,A -85,B 0,C 180,E1 -1680.502,E2 -1680.502} C_VEL
LIN {X 0,Y 580.056,Z 861.627,A -85,B 0,C 180,E1 -1681.803,E2 -1681.803} C_VEL
LIN {X 0,Y 580.059,Z 863.488,A -85,B 0,C 180,E1 -1682.588,E2 -1682.588} C_VEL
LIN {X 0,Y 580.045,Z 865.253,A -85,B 0,C 180,E1 -1683.716,E2 -1683.716} C_VEL
LIN {X 0,Y 580.021,Z 865.976,A -85,B 0,C 180,E1 -1684.908,E2 -1684.908} C_VEL
LIN {X 0,Y 580.026,Z 865.829,A -85,B 0,C 180,E1 -1685.673,E2 -1685.673} C_VEL
LIN {X 0,Y 580.047,Z 864.324,A -85,B 0,C 180,E1 -1687.05,E2 -1687.05} C_VEL
LIN {X 0,Y 580.078,Z 861.555,A -85,B 0,C 180,E1 -1688.315,E2 -1688.315} C_VEL
LIN {X 0,Y 580.109,Z 857.892,A -85,B 0,C 180,E1 -1689.432,E2 -1689.432} C_VEL
LIN {X 0,Y 580.15,Z 853.013,A -85,B 0,C 180,E1 -1690.542,E2 -1690.542} C_VEL
LIN {X 0,Y 580.177,Z 846.802,A -85,B 0,C 180,E1 -1691.643,E2 -1691.643} C_VEL
LIN {X 0,Y 580.199,Z 839.057,A -85,B 0,C 180,E1 -1692.737,E2 -1692.737} C_VEL
LIN {X 0,Y 580.277,Z 831.098,A -85,B 0,C 180,E1 -1693.646,E2 -1693.646} C_VEL
LIN {X 0,Y 580.313,Z 821.526,A -85,B 0,C 180,E1 -1694.549,E2 -1694.549} C_VEL
LIN {X 0,Y 580.432,Z 810.925,A -85,B 0,C 180,E1 -1695.352,E2 -1695.352} C_VEL
LIN {X 0,Y 580.562,Z 798.829,A -85,B 0,C 180,E1 -1696.079,E2 -1696.079} C_VEL
LIN {X 0,Y 580.676,Z 786.018,A -85,B 0,C 180,E1 -1696.662,E2 -1696.662} C_VEL
LIN {X 0,Y 580.742,Z 773.214,A -85,B 0,C 180,E1 -1697.086,E2 -1697.086} C_VEL
LIN {X 0,Y 580.811,Z 760.924,A -85,B 0,C 180,E1 -1697.354,E2 -1697.354} C_VEL
LIN {X 0,Y 580.888,Z 682.562,A -85,B 0,C 180,E1 -1698.337,E2 -1698.337} C_VEL
LIN {X 0,Y 580.384,Z 680.763,A -85,B 0,C 180,E1 -1698.415,E2 -1698.415} C_VEL
LIN {X 0,Y 580.293,Z 680.221,A -85,B 0,C 180,E1 -1698.571,E2 -1698.571} C_VEL
LIN {X 0,Y 580.303,Z 680.2,A -85,B 0,C 180,E1 -1701.645,E2 -1701.645} C_VEL
LIN {X 0,Y 580.297,Z 680.199,A -85,B 0,C 180,E1 -1704.441,E2 -1704.441} C_VEL
LIN {X 0,Y 580.304,Z 680.194,A -85,B 0,C 180,E1 -1707.224,E2 -1707.224} C_VEL
LIN {X 0,Y 580.351,Z 680.195,A -85,B 0,C 180,E1 -1710.001,E2 -1710.001} C_VEL
LIN {X 0,Y 580.312,Z 680.196,A -85,B 0,C 180,E1 -1712.778,E2 -1712.778} C_VEL
LIN {X 0,Y 580.287,Z 680.196,A -85,B 0,C 180,E1 -1715.561,E2 -1715.561} C_VEL
LIN {X 0,Y 580.292,Z 680.203,A -85,B 0,C 180,E1 -1718.358,E2 -1718.358} C_VEL
LIN {X 0,Y 580.274,Z 680.199,A -85,B 0,C 180,E1 -1721.175,E2 -1721.175} C_VEL
LIN {X 0,Y 580.293,Z 680.196,A -85,B 0,C 180,E1 -1724.019,E2 -1724.019} C_VEL
LIN {X 0,Y 580.274,Z 680.206,A -85,B 0,C 180,E1 -1726.899,E2 -1726.899} C_VEL
LIN {X 0,Y 580.258,Z 680.197,A -85,B 0,C 180,E1 -1729.825,E2 -1729.825} C_VEL
LIN {X 0,Y 580.246,Z 680.2,A -85,B 0,C 180,E1 -1732.055,E2 -1732.055} C_VEL
LIN {X 0,Y 580.244,Z 680.206,A -85,B 0,C 180,E1 -1734.712,E2 -1734.712} C_VEL
LIN {X 0,Y 580.249,Z 680.204,A -85,B 0,C 180,E1 -1737.405,E2 -1737.405} C_VEL
LIN {X 0,Y 580.233,Z 680.204,A -85,B 0,C 180,E1 -1739.777,E2 -1739.777} C_VEL
LIN {X 0,Y 580.274,Z 680.196,A -85,B 0,C 180,E1 -1742.203,E2 -1742.203} C_VEL
LIN {X 0,Y 580.257,Z 680.198,A -85,B 0,C 180,E1 -1744.699,E2 -1744.699} C_VEL
LIN {X 0,Y 580.269,Z 680.205,A -85,B 0,C 180,E1 -1747.272,E2 -1747.272} C_VEL
LIN {X 0,Y 580.242,Z 680.201,A -85,B 0,C 180,E1 -1750.264,E2 -1750.264} C_VEL
LIN {X 0,Y 580.216,Z 680.204,A -85,B 0,C 180,E1 -1752.713,E2 -1752.713} C_VEL
LIN {X 0,Y 580.234,Z 680.213,A -85,B 0,C 180,E1 -1755.614,E2 -1755.614} C_VEL
LIN {X 0,Y 580.233,Z 680.205,A -85,B 0,C 180,E1 -1758.227,E2 -1758.227} C_VEL
LIN {X 0,Y 580.239,Z 680.202,A -85,B 0,C 180,E1 -1760.962,E2 -1760.962} C_VEL
LIN {X 0,Y 580.211,Z 680.211,A -85,B 0,C 180,E1 -1763.592,E2 -1763.592} C_VEL
LIN {X 0,Y 580.264,Z 680.207,A -85,B 0,C 180,E1 -1766.141,E2 -1766.141} C_VEL
LIN {X 0,Y 580.239,Z 680.205,A -85,B 0,C 180,E1 -1768.612,E2 -1768.612} C_VEL
LIN {X 0,Y 580.243,Z 680.203,A -85,B 0,C 180,E1 -1771.021,E2 -1771.021} C_VEL
LIN {X 0,Y 580.307,Z 680.347,A -85,B 0,C 180,E1 -1773.604,E2 -1773.604} C_VEL
LIN {X 0,Y 580.488,Z 681.271,A -85,B 0,C 180,E1 -1773.715,E2 -1773.715} C_VEL
LIN {X 0,Y 580.9,Z 682.521,A -85,B 0,C 180,E1 -1773.753,E2 -1773.753} C_VEL
LIN {X 0,Y 580.784,Z 761.744,A -85,B 0,C 180,E1 -1774.751,E2 -1774.751} C_VEL
LIN {X 0,Y 580.733,Z 774.201,A -85,B 0,C 180,E1 -1775.035,E2 -1775.035} C_VEL
LIN {X 0,Y 580.648,Z 785.674,A -85,B 0,C 180,E1 -1775.417,E2 -1775.417} C_VEL
LIN {X 0,Y 580.588,Z 796.293,A -85,B 0,C 180,E1 -1775.886,E2 -1775.886} C_VEL
LIN {X 0,Y 580.499,Z 806.446,A -85,B 0,C 180,E1 -1776.451,E2 -1776.451} C_VEL
LIN {X 0,Y 580.394,Z 816.277,A -85,B 0,C 180,E1 -1777.125,E2 -1777.125} C_VEL
LIN {X 0,Y 580.312,Z 826.094,A -85,B 0,C 180,E1 -1777.949,E2 -1777.949} C_VEL
LIN {X 0,Y 580.246,Z 835.556,A -85,B 0,C 180,E1 -1778.929,E2 -1778.929} C_VEL
LIN {X 0,Y 580.171,Z 843.779,A -85,B 0,C 180,E1 -1779.988,E2 -1779.988} C_VEL
LIN {X 0,Y 580.142,Z 849.582,A -85,B 0,C 180,E1 -1780.908,E2 -1780.908} C_VEL
LIN {X 0,Y 580.09,Z 855.167,A -85,B 0,C 180,E1 -1782.004,E2 -1782.004} C_VEL
LIN {X 0,Y 580.058,Z 859.693,A -85,B 0,C 180,E1 -1783.172,E2 -1783.172} C_VEL
LIN {X 0,Y 580.068,Z 861.673,A -85,B 0,C 180,E1 -1783.819,E2 -1783.819} C_VEL
LIN {X 0,Y 580.032,Z 863.384,A -85,B 0,C 180,E1 -1784.54,E2 -1784.54} C_VEL
LIN {X 0,Y 580.054,Z 865.306,A -85,B 0,C 180,E1 -1785.766,E2 -1785.766} C_VEL
LIN {X 0,Y 580.061,Z 865.927,A -85,B 0,C 180,E1 -1786.691,E2 -1786.691} C_VEL
LIN {X 0,Y 580.05,Z 865.926,A -85,B 0,C 180,E1 -1787.403,E2 -1787.403} C_VEL
LIN {X 0,Y 580.055,Z 865.531,A -85,B 0,C 180,E1 -1788.113,E2 -1788.113} C_VEL
LIN {X 0,Y 580.076,Z 864.523,A -85,B 0,C 180,E1 -1788.925,E2 -1788.925} C_VEL
LIN {X 0,Y 580.062,Z 861.767,A -85,B 0,C 180,E1 -1790.234,E2 -1790.234} C_VEL
LIN {X 0,Y 580.089,Z 858.412,A -85,B 0,C 180,E1 -1791.289,E2 -1791.289} C_VEL
LIN {X 0,Y 580.114,Z 853.986,A -85,B 0,C 180,E1 -1792.342,E2 -1792.342} C_VEL
LIN {X 0,Y 580.139,Z 847.331,A -85,B 0,C 180,E1 -1793.559,E2 -1793.559} C_VEL
LIN {X 0,Y 580.164,Z 840.006,A -85,B 0,C 180,E1 -1794.613,E2 -1794.613} C_VEL
LIN {X 0,Y 580.28,Z 832.598,A -85,B 0,C 180,E1 -1795.485,E2 -1795.485} C_VEL
LIN {X 0,Y 580.33,Z 823.722,A -85,B 0,C 180,E1 -1796.355,E2 -1796.355} C_VEL
LIN {X 0,Y 580.426,Z 813.971,A -85,B 0,C 180,E1 -1797.137,E2 -1797.137} C_VEL
LIN {X 0,Y 580.524,Z 803.299,A -85,B 0,C 180,E1 -1797.832,E2 -1797.832} C_VEL
LIN {X 0,Y 580.613,Z 791.382,A -85,B 0,C 180,E1 -1798.439,E2 -1798.439} C_VEL
LIN {X 0,Y 580.739,Z 778.17,A -85,B 0,C 180,E1 -1798.938,E2 -1798.938} C_VEL
LIN {X 0,Y 580.778,Z 765.622,A -85,B 0,C 180,E1 -1799.263,E2 -1799.263} C_VEL
LIN {X 0,Y 580.842,Z 751.653,A -85,B 0,C 180,E1 -1799.48,E2 -1799.48} C_VEL
LIN {X 0,Y 580.802,Z 682.176,A -85,B 0,C 180,E1 -1800.347,E2 -1800.347} C_VEL
LIN {X 0,Y 580.412,Z 680.606,A -85,B 0,C 180,E1 -1800.434,E2 -1800.434} C_VEL
LIN {X 0,Y 580.355,Z 680.202,A -85,B 0,C 180,E1 -1800.607,E2 -1800.607} C_VEL
LIN {X 0,Y 580.335,Z 680.192,A -85,B 0,C 180,E1 -1802.776,E2 -1802.776} C_VEL
LIN {X 0,Y 580.325,Z 680.195,A -85,B 0,C 180,E1 -1805.56,E2 -1805.56} C_VEL
LIN {X 0,Y 580.314,Z 680.2,A -85,B 0,C 180,E1 -1808.356,E2 -1808.356} C_VEL
LIN {X 0,Y 580.308,Z 680.193,A -85,B 0,C 180,E1 -1811.191,E2 -1811.191} C_VEL
LIN {X 0,Y 580.33,Z 680.196,A -85,B 0,C 180,E1 -1814.017,E2 -1814.017} C_VEL
LIN {X 0,Y 580.32,Z 680.194,A -85,B 0,C 180,E1 -1816.914,E2 -1816.914} C_VEL
LIN {X 0,Y 580.291,Z 680.196,A -85,B 0,C 180,E1 -1819.823,E2 -1819.823} C_VEL
LIN {X 0,Y 580.272,Z 680.2,A -85,B 0,C 180,E1 -1822.053,E2 -1822.053} C_VEL
LIN {X 0,Y 580.307,Z 680.197,A -85,B 0,C 180,E1 -1825.08,E2 -1825.08} C_VEL
LIN {X 0,Y 580.287,Z 680.198,A -85,B 0,C 180,E1 -1828.186,E2 -1828.186} C_VEL
LIN {X 0,Y 580.289,Z 680.203,A -85,B 0,C 180,E1 -1830.694,E2 -1830.694} C_VEL
LIN {X 0,Y 580.288,Z 680.2,A -85,B 0,C 180,E1 -1833.313,E2 -1833.313} C_VEL
LIN {X 0,Y 580.25,Z 680.201,A -85,B 0,C 180,E1 -1835.756,E2 -1835.756} C_VEL
LIN {X 0,Y 580.291,Z 680.195,A -85,B 0,C 180,E1 -1838.146,E2 -1838.146} C_VEL
LIN {X 0,Y 580.301,Z 680.199,A -85,B 0,C 180,E1 -1840.843,E2 -1840.843} C_VEL
LIN {X 0,Y 580.279,Z 680.201,A -85,B 0,C 180,E1 -1843.658,E2 -1843.658} C_VEL
LIN {X 0,Y 580.279,Z 680.197,A -85,B 0,C 180,E1 -1846.609,E2 -1846.609} C_VEL
LIN {X 0,Y 580.301,Z 680.199,A -85,B 0,C 180,E1 -1849.156,E2 -1849.156} C_VEL
LIN {X 0,Y 580.291,Z 680.199,A -85,B 0,C 180,E1 -1851.927,E2 -1851.927} C_VEL
LIN {X 0,Y 580.254,Z 680.2,A -85,B 0,C 180,E1 -1854.452,E2 -1854.452} C_VEL
LIN {X 0,Y 580.294,Z 680.196,A -85,B 0,C 180,E1 -1856.974,E2 -1856.974} C_VEL
LIN {X 0,Y 580.3,Z 680.2,A -85,B 0,C 180,E1 -1859.424,E2 -1859.424} C_VEL
LIN {X 0,Y 580.265,Z 680.209,A -85,B 0,C 180,E1 -1862.148,E2 -1862.148} C_VEL
LIN {X 0,Y 580.308,Z 680.407,A -85,B 0,C 180,E1 -1862.891,E2 -1862.891} C_VEL
LIN {X 0,Y 581.689,Z 686.064,A -85,B 0,C 180,E1 -1863.627,E2 -1863.627} C_VEL
LIN {X 0,Y 581.417,Z 708.017,A -85,B 0,C 180,E1 -1866.112,E2 -1866.112} C_VEL
LIN {X 0,Y 581.083,Z 736.594,A -85,B 0,C 180,E1 -1869.281,E2 -1869.281} C_VEL
LIN {X 0,Y 580.821,Z 761.809,A -85,B 0,C 180,E1 -1872.027,E2 -1872.027} C_VEL
LIN {X 0,Y 580.602,Z 788.705,A -85,B 0,C 180,E1 -1874.914,E2 -1874.914} C_VEL
LIN {X 0,Y 580.51,Z 801.876,A -85,B 0,C 180,E1 -1876.299,E2 -1876.299} C_VEL
LIN {X 0,Y 580.945,Z 805.854,A -85,B 0,C 180,E1 -1876.377,E2 -1876.377} C_VEL
LIN {X 0,Y 580.799,Z 911.896,A -85,B 0,C 180,E1 -1877.707,E2 -1877.707} C_VEL
LIN {X 0,Y 580.754,Z 925.185,A -85,B 0,C 180,E1 -1878.016,E2 -1878.016} C_VEL
LIN {X 0,Y 580.659,Z 937.346,A -85,B 0,C 180,E1 -1878.435,E2 -1878.435} C_VEL
LIN {X 0,Y 580.564,Z 949.614,A -85,B 0,C 180,E1 -1879.008,E2 -1879.008} C_VEL
LIN {X 0,Y 580.441,Z 961.187,A -85,B 0,C 180,E1 -1879.711,E2 -1879.711} C_VEL
LIN {X 0,Y 580.343,Z 971.586,A -85,B 0,C 180,E1 -1880.502,E2 -1880.502} C_VEL
LIN {X 0,Y 580.263,Z 980.027,A -85,B 0,C 180,E1 -1881.291,E2 -1881.291} C_VEL
LIN {X 0,Y 580.222,Z 987.952,A -85,B 0,C 180,E1 -1882.167,E2 -1882.167} C_VEL
LIN {X 0,Y 580.157,Z 995.63,A -85,B 0,C 180,E1 -1883.219,E2 -1883.219} C_VEL
LIN {X 0,Y 580.139,Z 1002.675,A -85,B 0,C 180,E1 -1884.437,E2 -1884.437} C_VEL
LIN {X 0,Y 580.108,Z 1007.367,A -85,B 0,C 180,E1 -1885.482,E2 -1885.482} C_VEL
LIN {X 0,Y 580.123,Z 1010.953,A -85,B 0,C 180,E1 -1886.526,E2 -1886.526} C_VEL
LIN {X 0,Y 580.043,Z 1012.806,A -85,B 0,C 180,E1 -1887.221,E2 -1887.221} C_VEL
LIN {X 0,Y 580.038,Z 1014.199,A -85,B 0,C 180,E1 -1887.916,E2 -1887.916} C_VEL
LIN {X 0,Y 580.04,Z 1015.784,A -85,B 0,C 180,E1 -1889.305,E2 -1889.305} C_VEL
LIN {X 0,Y 580.037,Z 1016,A -85,B 0,C 180,E1 -1889.999,E2 -1889.999} C_VEL
LIN {X 0,Y 580.046,Z 1015.186,A -85,B 0,C 180,E1 -1891.388,E2 -1891.388} C_VEL
LIN {X 0,Y 580.038,Z 1014.203,A -85,B 0,C 180,E1 -1892.082,E2 -1892.082} C_VEL
LIN {X 0,Y 580.043,Z 1012.812,A -85,B 0,C 180,E1 -1892.777,E2 -1892.777} C_VEL
LIN {X 0,Y 580.109,Z 1009.899,A -85,B 0,C 180,E1 -1893.82,E2 -1893.82} C_VEL
LIN {X 0,Y 580.053,Z 1005.954,A -85,B 0,C 180,E1 -1894.864,E2 -1894.864} C_VEL
LIN {X 0,Y 580.14,Z 999.884,A -85,B 0,C 180,E1 -1896.084,E2 -1896.084} C_VEL
LIN {X 0,Y 580.183,Z 993.244,A -85,B 0,C 180,E1 -1897.131,E2 -1897.131} C_VEL
LIN {X 0,Y 580.246,Z 984.999,A -85,B 0,C 180,E1 -1898.181,E2 -1898.181} C_VEL
LIN {X 0,Y 580.332,Z 974.613,A -85,B 0,C 180,E1 -1899.233,E2 -1899.233} C_VEL
LIN {X 0,Y 580.43,Z 964.944,A -85,B 0,C 180,E1 -1900.023,E2 -1900.023} C_VEL
LIN {X 0,Y 580.534,Z 954.346,A -85,B 0,C 180,E1 -1900.726,E2 -1900.726} C_VEL
LIN {X 0,Y 580.646,Z 942.099,A -85,B 0,C 180,E1 -1901.36,E2 -1901.36} C_VEL
LIN {X 0,Y 580.693,Z 930.209,A -85,B 0,C 180,E1 -1901.828,E2 -1901.828} C_VEL
LIN {X 0,Y 580.757,Z 917.569,A -85,B 0,C 180,E1 -1902.181,E2 -1902.181} C_VEL
LIN {X 0,Y 580.858,Z 904.402,A -85,B 0,C 180,E1 -1902.4,E2 -1902.4} C_VEL
LIN {X 0,Y 580.832,Z 804.236,A -85,B 0,C 180,E1 -1903.646,E2 -1903.646} C_VEL
LIN {X 0,Y 580.506,Z 801.65,A -85,B 0,C 180,E1 -1903.721,E2 -1903.721} C_VEL
LIN {X 0,Y 580.71,Z 775.277,A -85,B 0,C 180,E1 -1906.522,E2 -1906.522} C_VEL
LIN {X 0,Y 580.98,Z 747.745,A -85,B 0,C 180,E1 -1909.499,E2 -1909.499} C_VEL
LIN {X 0,Y 581.202,Z 723.166,A -85,B 0,C 180,E1 -1912.201,E2 -1912.201} C_VEL
LIN {X 0,Y 581.419,Z 703.137,A -85,B 0,C 180,E1 -1914.439,E2 -1914.439} C_VEL
LIN {X 0,Y 581.686,Z 686.07,A -85,B 0,C 180,E1 -1916.372,E2 -1916.372} C_VEL
LIN {X 0,Y 580.301,Z 680.328,A -85,B 0,C 180,E1 -1917.131,E2 -1917.131} C_VEL
LIN {X 0,Y 580.283,Z 680.203,A -85,B 0,C 180,E1 -1919.772,E2 -1919.772} C_VEL
LIN {X 0,Y 580.295,Z 680.203,A -85,B 0,C 180,E1 -1922.199,E2 -1922.199} C_VEL
LIN {X 0,Y 580.283,Z 680.202,A -85,B 0,C 180,E1 -1924.695,E2 -1924.695} C_VEL
LIN {X 0,Y 580.292,Z 680.195,A -85,B 0,C 180,E1 -1927.267,E2 -1927.267} C_VEL
LIN {X 0,Y 580.285,Z 680.201,A -85,B 0,C 180,E1 -1930.269,E2 -1930.269} C_VEL
LIN {X 0,Y 580.271,Z 680.207,A -85,B 0,C 180,E1 -1932.705,E2 -1932.705} C_VEL
LIN {X 0,Y 580.267,Z 680.198,A -85,B 0,C 180,E1 -1935.608,E2 -1935.608} C_VEL
LIN {X 0,Y 580.306,Z 680.195,A -85,B 0,C 180,E1 -1938.233,E2 -1938.233} C_VEL
LIN {X 0,Y 580.283,Z 680.206,A -85,B 0,C 180,E1 -1940.965,E2 -1940.965} C_VEL
LIN {X 0,Y 580.288,Z 680.196,A -85,B 0,C 180,E1 -1943.598,E2 -1943.598} C_VEL
LIN {X 0,Y 580.311,Z 680.192,A -85,B 0,C 180,E1 -1946.145,E2 -1946.145} C_VEL
LIN {X 0,Y 580.268,Z 680.199,A -85,B 0,C 180,E1 -1948.614,E2 -1948.614} C_VEL
LIN {X 0,Y 580.286,Z 680.201,A -85,B 0,C 180,E1 -1951.023,E2 -1951.023} C_VEL
LIN {X 0,Y 580.317,Z 680.198,A -85,B 0,C 180,E1 -1953.658,E2 -1953.658} C_VEL
LIN {X 0,Y 580.27,Z 680.197,A -85,B 0,C 180,E1 -1956.442,E2 -1956.442} C_VEL
LIN {X 0,Y 580.265,Z 680.205,A -85,B 0,C 180,E1 -1959.437,E2 -1959.437} C_VEL
LIN {X 0,Y 580.268,Z 680.208,A -85,B 0,C 180,E1 -1961.645,E2 -1961.645} C_VEL
LIN {X 0,Y 580.263,Z 680.209,A -85,B 0,C 180,E1 -1963.825,E2 -1963.825} C_VEL
LIN {X 0,Y 580.315,Z 680.2,A -85,B 0,C 180,E1 -1965.983,E2 -1965.983} C_VEL
